KUKA KRL program: MyProgram_030().src

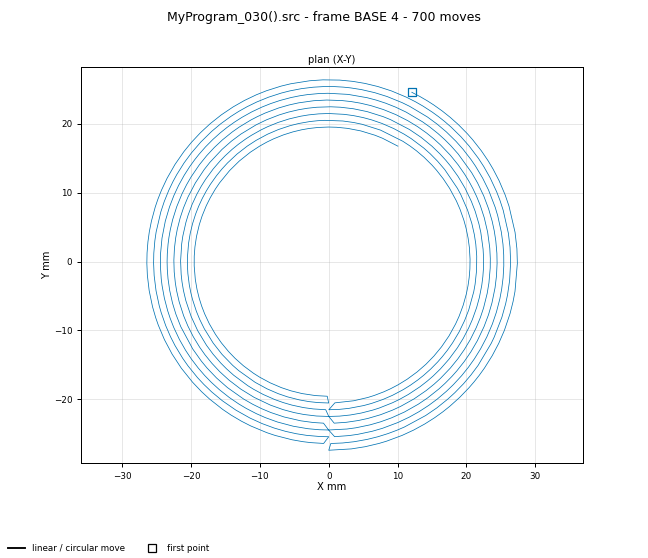
[picture p0: tool path of MyProgram_030().src in frame BASE 4, 700 of 700 moves have a stored position in this frame; points joined in program order, loops and branches not executed]
&ACCESS RVP
&REL 1
&PARAM TEMPLATE = C:\KRC\Roboter\Template\vorgabe
&PARAM EDITMASK = *
DEF MyProgram_030()
; ---- Setting reference (Base) ----
$BASE = BASE_DATA[4]

; --------------------------
; ---- Setting tool (TCP) ----
$TOOL = TOOL_DATA[3]
; --------------------------

$VEL.CP = VEL_APROX_PRINT
Startdeposition()
$VEL.CP = VEL_PRINT
LIN {X 12.0703,Y 24.5921,Z 59,A 55.5267,B 24.8071,C -3.2024,E1 25.0724,E2 -692.837} C_DIS
LIN {X 13.2585,Y 23.9727,Z 59,A 52.8062,B 24.8075,C -3.1996,E1 25.0791,E2 -690.1175} C_DIS
LIN {X 14.3009,Y 23.3657,Z 59,A 50.2739,B 24.8079,C -3.1959,E1 25.0852,E2 -687.5843} C_DIS
LIN {X 15.2376,Y 22.7662,Z 59,A 47.9776,B 24.8083,C -3.1926,E1 25.0906,E2 -685.2878} C_DIS
LIN {X 16.4743,Y 21.887,Z 59,A 44.3349,B 24.8096,C -3.1823,E1 25.0988,E2 -681.6335} C_DIS
LIN {X 17.6466,Y 20.9541,Z 59,A 41.1874,B 24.8103,C -3.1764,E1 25.1056,E2 -678.484} C_DIS
LIN {X 18.834,Y 19.8936,Z 59,A 38.0345,B 24.8108,C -3.1718,E1 25.112,E2 -675.333} C_DIS
LIN {X 20.1281,Y 18.5822,Z 59,A 34.6982,B 24.8111,C -3.1694,E1 25.1185,E2 -672.0053} C_DIS
LIN {X 20.8979,Y 17.7129,Z 59,A 31.723,B 24.8125,C -3.1578,E1 25.1239,E2 -669.0162} C_DIS
LIN {X 22.1576,Y 16.1093,Z 59,A 27.8177,B 24.8132,C -3.1518,E1 25.1305,E2 -665.1153} C_DIS
LIN {X 23.1629,Y 14.6275,Z 59,A 23.876,B 24.8146,C -3.1402,E1 25.1366,E2 -661.1657} C_DIS
LIN {X 23.8751,Y 13.4329,Z 59,A 20.9616,B 24.8155,C -3.1326,E1 25.1406,E2 -658.2484} C_DIS
LIN {X 24.7489,Y 11.7454,Z 59,A 16.9906,B 24.8168,C -3.1219,E1 25.1455,E2 -654.2731} C_DIS
LIN {X 25.6294,Y 9.6744,Z 59,A 11.8386,B 24.8189,C -3.1034,E1 25.1509,E2 -649.1059} C_DIS
LIN {X 26.1818,Y 8.0609,Z 59,A 7.6845,B 24.8209,C -3.0861,E1 25.1543,E2 -644.9344} C_DIS
LIN {X 27.0615,Y 4.2601,Z 59,A 1.2889,B 24.8214,C -3.0826,E1 25.158,E2 -638.5678} C_DIS
LIN {X 27.3301,Y 1.8802,Z 59,A -5.3272,B 24.8254,C -3.0478,E1 25.1597,E2 -631.9085} C_DIS
LIN {X 27.3946,Y -0.2461,Z 59,A -10.1009,B 24.8274,C -3.0301,E1 25.1596,E2 -627.1211} C_DIS
LIN {X 27.0526,Y -4.3175,Z 59,A -16.9925,B 24.8282,C -3.0233,E1 25.1575,E2 -620.2542} C_DIS
LIN {X 26.776,Y -5.7881,Z 59,A -20.1318,B 24.8293,C -3.0135,E1 25.1557,E2 -617.11} C_DIS
LIN {X 26.3337,Y -7.5501,Z 59,A -23.8827,B 24.8306,C -3.0024,E1 25.153,E2 -613.3544} C_DIS
LIN {X 25.5178,Y -9.9656,Z 59,A -30.3379,B 24.8339,C -2.973,E1 25.1468,E2 -606.8657} C_DIS
LIN {X 24.6926,Y -11.8634,Z 59,A -33.9623,B 24.8344,C -2.9686,E1 25.1426,E2 -603.2505} C_DIS
LIN {X 23.7431,Y -13.6635,Z 59,A -37.9233,B 24.8353,C -2.9601,E1 25.1372,E2 -599.2899} C_DIS
LIN {X 22.6158,Y -15.4593,Z 59,A -41.7608,B 24.8359,C -2.9549,E1 25.1314,E2 -595.4595} C_DIS
LIN {X 21.8598,Y -16.5112,Z 59,A -44.5998,B 24.8369,C -2.9462,E1 25.1267,E2 -592.6136} C_DIS
LIN {X 21.1214,Y -17.4459,Z 59,A -47.2368,B 24.8378,C -2.9381,E1 25.1221,E2 -589.9696} C_DIS
LIN {X 20.3552,Y -18.3341,Z 59,A -49.8939,B 24.8387,C -2.9297,E1 25.1172,E2 -587.3044} C_DIS
LIN {X 18.9974,Y -19.7374,Z 59,A -54.0497,B 24.8399,C -2.9192,E1 25.1089,E2 -583.1413} C_DIS
LIN {X 17.5559,Y -21.03,Z 59,A -57.5749,B 24.8402,C -2.9161,E1 25.1015,E2 -579.6227} C_DIS
LIN {X 16.5729,Y -21.8133,Z 59,A -60.5172,B 24.8412,C -2.9071,E1 25.095,E2 -576.6699} C_DIS
LIN {X 15.3797,Y -22.6701,Z 59,A -63.5679,B 24.8418,C -2.9013,E1 25.088,E2 -573.6159} C_DIS
LIN {X 13.9552,Y -23.5737,Z 59,A -67.0294,B 24.8425,C -2.8956,E1 25.0798,E2 -570.1517} C_DIS
LIN {X 12.3253,Y -24.4654,Z 59,A -71.4342,B 24.8438,C -2.8836,E1 25.0689,E2 -565.7309} C_DIS
LIN {X 10.6544,Y -25.2378,Z 59,A -75.2339,B 24.8443,C -2.8786,E1 25.0591,E2 -561.9284} C_DIS
LIN {X 8.4028,Y -26.0738,Z 59,A -79.4966,B 24.8442,C -2.8801,E1 25.0479,E2 -557.6779} C_DIS
LIN {X 7.3143,Y -26.4001,Z 59,A -82.2216,B 24.8448,C -2.874,E1 25.0406,E2 -554.943} C_DIS
LIN {X 5.3186,Y -26.8736,Z 59,A -86.9065,B 24.8456,C -2.8663,E1 25.0278,E2 -550.246} C_DIS
LIN {X 3.2945,Y -27.1959,Z 59,A -91.5499,B 24.8463,C -2.8601,E1 25.0149,E2 -545.5918} C_DIS
LIN {X 0.0059,Y -27.3922,Z 59,A -95.1262,B 24.8432,C -2.889,E1 25.0051,E2 -542.0856} C_DIS
Enddeposition()
LIN {X 0.0059,Y -27.3922,Z 59,A -95.1262,B 24.8432,C -2.889,E1 25.0051,E2 -542.0856} C_DIS
Startdeposition()
$VEL.CP = VEL_PRINT
LIN {X 0.2993,Y -26.4122,Z 59,A -95.4906,B 24.8424,C -2.8963,E1 25.0042,E2 -541.7387} C_DIS
LIN {X 2.0234,Y -26.3363,Z 59,A -91.3024,B 24.8418,C -2.902,E1 25.0159,E2 -545.9388} C_DIS
LIN {X 3.7058,Y -26.1526,Z 59,A -87.6758,B 24.8415,C -2.9039,E1 25.0259,E2 -549.5669} C_DIS
LIN {X 5.5925,Y -25.8151,Z 59,A -83.5455,B 24.8412,C -2.9071,E1 25.0372,E2 -553.6998} C_DIS
LIN {X 7.1324,Y -25.4327,Z 59,A -80.3986,B 24.8412,C -2.9077,E1 25.0457,E2 -556.8432} C_DIS
LIN {X 8.5837,Y -24.9799,Z 59,A -77.2197,B 24.8408,C -2.9104,E1 25.0541,E2 -560.0224} C_DIS
LIN {X 9.8795,Y -24.4969,Z 59,A -74.2469,B 24.8404,C -2.9141,E1 25.0619,E2 -562.9976} C_DIS
LIN {X 10.9902,Y -24.019,Z 59,A -70.5185,B 24.8387,C -2.9297,E1 25.0714,E2 -566.7536} C_DIS
LIN {X 14.0844,Y -22.3457,Z 59,A -63.6414,B 24.8381,C -2.9349,E1 25.088,E2 -573.6223} C_DIS
LIN {X 15.6927,Y -21.2472,Z 59,A -59.3824,B 24.8372,C -2.9437,E1 25.0977,E2 -577.8875} C_DIS
LIN {X 17.2836,Y -19.9745,Z 59,A -55.1439,B 24.8363,C -2.9513,E1 25.1068,E2 -582.1276} C_DIS
LIN {X 18.3176,Y -19.0305,Z 59,A -51.8874,B 24.8353,C -2.9608,E1 25.1135,E2 -585.3932} C_DIS
LIN {X 19.5777,Y -17.7319,Z 59,A -48.5226,B 24.8349,C -2.9639,E1 25.1199,E2 -588.7508} C_DIS
LIN {X 20.6509,Y -16.4691,Z 59,A -44.3687,B 24.8332,C -2.9795,E1 25.1273,E2 -592.9225} C_DIS
LIN {X 21.6906,Y -15.0734,Z 59,A -39.8108,B 24.831,C -2.9989,E1 25.1346,E2 -597.5039} C_DIS
LIN {X 23.5983,Y -11.8668,Z 59,A -33.2485,B 24.8304,C -3.0036,E1 25.1435,E2 -604.0433} C_DIS
LIN {X 24.0437,Y -10.9355,Z 59,A -29.9775,B 24.8283,C -3.0224,E1 25.1474,E2 -607.3412} C_DIS
LIN {X 25.1471,Y -8.0821,Z 59,A -23.9084,B 24.8268,C -3.0356,E1 25.1531,E2 -613.4073} C_DIS
LIN {X 25.6939,Y -6.1255,Z 59,A -20.1339,B 24.8261,C -3.0415,E1 25.1558,E2 -617.1743} C_DIS
LIN {X 25.9662,Y -4.8406,Z 59,A -17.0738,B 24.8248,C -3.0529,E1 25.1574,E2 -620.2434} C_DIS
LIN {X 26.2688,Y -2.7644,Z 59,A -11.7155,B 24.822,C -3.0768,E1 25.1593,E2 -625.6269} C_DIS
LIN {X 26.4161,Y -0.0885,Z 59,A -6.3971,B 24.8206,C -3.089,E1 25.1598,E2 -630.9423} C_DIS
LIN {X 26.3302,Y 2.1008,Z 59,A -1.385,B 24.8185,C -3.1069,E1 25.1589,E2 -635.967} C_DIS
LIN {X 26.0901,Y 4.1243,Z 59,A 3.4136,B 24.8164,C -3.1249,E1 25.1569,E2 -640.7802} C_DIS
LIN {X 25.3421,Y 7.4472,Z 59,A 9.6225,B 24.8155,C -3.1328,E1 25.1528,E2 -646.9719} C_DIS
LIN {X 24.8708,Y 8.8956,Z 59,A 13.13,B 24.814,C -3.1447,E1 25.1496,E2 -650.4879} C_DIS
LIN {X 24.3916,Y 10.136,Z 59,A 16.1141,B 24.8129,C -3.154,E1 25.1465,E2 -653.4776} C_DIS
LIN {X 23.4463,Y 12.1643,Z 59,A 21.2351,B 24.811,C -3.1702,E1 25.1401,E2 -658.6096} C_DIS
LIN {X 22.5009,Y 13.8356,Z 59,A 25.1058,B 24.8101,C -3.1776,E1 25.1346,E2 -662.4779} C_DIS
LIN {X 21.7431,Y 14.9976,Z 59,A 28.195,B 24.8091,C -3.1859,E1 25.1298,E2 -665.5716} C_DIS
LIN {X 20.3882,Y 16.7935,Z 59,A 32.3345,B 24.8087,C -3.189,E1 25.1227,E2 -669.6989} C_DIS
LIN {X 19.2048,Y 18.1348,Z 59,A 37.0991,B 24.8065,C -3.2072,E1 25.1137,E2 -674.4856} C_DIS
LIN {X 17.7872,Y 19.5274,Z 59,A 40.7472,B 24.8064,C -3.2086,E1 25.1063,E2 -678.1221} C_DIS
LIN {X 16.8166,Y 20.3691,Z 59,A 43.3718,B 24.806,C -3.2121,E1 25.1007,E2 -680.7447} C_DIS
LIN {X 15.9526,Y 21.0528,Z 59,A 45.8165,B 24.8054,C -3.2169,E1 25.0953,E2 -683.1917} C_DIS
LIN {X 15.0479,Y 21.7084,Z 59,A 48.563,B 24.8045,C -3.2242,E1 25.089,E2 -685.9461} C_DIS
LIN {X 13.6911,Y 22.5887,Z 59,A 51.7172,B 24.8043,C -3.2258,E1 25.0816,E2 -689.094} C_DIS
LIN {X 12.6011,Y 23.2143,Z 59,A 54.6274,B 24.8036,C -3.2313,E1 25.0745,E2 -692.0088} C_DIS
LIN {X 11.2915,Y 23.8787,Z 59,A 58.2581,B 24.8026,C -3.2396,E1 25.0653,E2 -695.6495} C_DIS
LIN {X 9.1052,Y 24.7944,Z 59,A 62.8093,B 24.8027,C -3.2388,E1 25.0536,E2 -700.1886} C_DIS
LIN {X 7.1428,Y 25.4295,Z 59,A 67.9203,B 24.8016,C -3.2481,E1 25.0399,E2 -705.3127} C_DIS
LIN {X 5.2719,Y 25.8825,Z 59,A 71.5741,B 24.8019,C -3.2452,E1 25.03,E2 -708.9548} C_DIS
LIN {X 3.4856,Y 26.183,Z 59,A 75.855,B 24.8014,C -3.2495,E1 25.0181,E2 -713.242} C_DIS
LIN {X 1.5804,Y 26.3662,Z 59,A 80.1393,B 24.8012,C -3.2508,E1 25.0062,E2 -717.5274} C_DIS
LIN {X -0.8248,Y 26.401,Z 59,A 85.1216,B 24.8016,C -3.2477,E1 24.9923,E2 -722.5021} C_DIS
LIN {X -2.7464,Y 26.2707,Z 59,A 89.7241,B 24.8014,C -3.2493,E1 24.9795,E2 -727.1108} C_DIS
LIN {X -5.5246,Y 25.8296,Z 59,A 94.8895,B 24.8029,C -3.2373,E1 24.9654,E2 -732.2526} C_DIS
LIN {X -6.9255,Y 25.4898,Z 59,A 98.7337,B 24.8026,C -3.2398,E1 24.9549,E2 -736.1086} C_DIS
LIN {X -9.0534,Y 24.8138,Z 59,A 103.2055,B 24.8036,C -3.2313,E1 24.9431,E2 -740.5684} C_DIS
LIN {X -10.5209,Y 24.2282,Z 59,A 106.666,B 24.8042,C -3.2268,E1 24.9342,E2 -744.0261} C_DIS
LIN {X -12.2342,Y 23.4094,Z 59,A 111.5552,B 24.8042,C -3.2259,E1 24.922,E2 -748.9262} C_DIS
LIN {X -13.8723,Y 22.4777,Z 59,A 115.2888,B 24.8055,C -3.2162,E1 24.9131,E2 -752.648} C_DIS
LIN {X -15.6046,Y 21.3117,Z 59,A 119.666,B 24.8067,C -3.2063,E1 24.9031,E2 -757.0166} C_DIS
LIN {X -17.2144,Y 20.034,Z 59,A 124.0536,B 24.8079,C -3.1963,E1 24.8937,E2 -761.397} C_DIS
LIN {X -18.6321,Y 18.7227,Z 59,A 128.3146,B 24.809,C -3.1872,E1 24.8851,E2 -765.6537} C_DIS
LIN {X -19.9447,Y 17.3177,Z 59,A 132.7337,B 24.81,C -3.1785,E1 24.8769,E2 -770.0719} C_DIS
LIN {X -21.0478,Y 15.9592,Z 59,A 136.4195,B 24.8113,C -3.1681,E1 24.8706,E2 -773.75} C_DIS
LIN {X -22.3201,Y 14.1253,Z 59,A 141.3942,B 24.8127,C -3.1558,E1 24.8629,E2 -778.7202} C_DIS
LIN {X -23.4768,Y 12.1054,Z 59,A 146.3251,B 24.8145,C -3.1408,E1 24.8563,E2 -783.6412} C_DIS
LIN {X -24.2947,Y 10.3665,Z 59,A 150.5155,B 24.8159,C -3.1287,E1 24.8515,E2 -787.8257} C_DIS
LIN {X -24.82,Y 9.0365,Z 59,A 153.5544,B 24.8171,C -3.1191,E1 24.8486,E2 -790.8587} C_DIS
LIN {X -25.2006,Y 7.9134,Z 59,A 156.3755,B 24.8178,C -3.1127,E1 24.8462,E2 -793.6808} C_DIS
LIN {X -25.7517,Y 5.875,Z 59,A 160.3956,B 24.8199,C -3.0955,E1 24.8434,E2 -797.683} C_DIS
LIN {X -26.0575,Y 4.3243,Z 59,A 163.709,B 24.8212,C -3.0842,E1 24.8417,E2 -800.989} C_DIS
LIN {X -26.2568,Y 2.8758,Z 59,A 167.4625,B 24.8219,C -3.0776,E1 24.8404,E2 -804.7491} C_DIS
LIN {X -26.3843,Y 1.2532,Z 59,A 170.8053,B 24.8233,C -3.0655,E1 24.8399,E2 -808.0831} C_DIS
LIN {X -26.4138,Y -0.2385,Z 59,A 174.1449,B 24.8244,C -3.056,E1 24.8399,E2 -811.42} C_DIS
LIN {X -26.3409,Y -1.9594,Z 59,A 178.5048,B 24.8254,C -3.0481,E1 24.8406,E2 -815.787} C_DIS
LIN {X -26.0758,Y -4.2115,Z 59,A -176.6427,B 24.8271,C -3.0327,E1 24.8425,E2 -820.6316} C_DIS
LIN {X -25.5842,Y -6.5683,Z 59,A -171.8967,B 24.8292,C -3.0142,E1 24.8455,E2 -825.3613} C_DIS
LIN {X -25.1234,Y -8.1552,Z 59,A -168.5165,B 24.8305,C -3.0026,E1 24.8482,E2 -828.7332} C_DIS
LIN {X -24.7509,Y -9.2239,Z 59,A -165.4952,B 24.831,C -2.999,E1 24.8511,E2 -831.7628} C_DIS
LIN {X -23.8641,Y -11.3221,Z 59,A -160.9304,B 24.8328,C -2.983,E1 24.8563,E2 -836.3145} C_DIS
LIN {X -22.7493,Y -13.4226,Z 59,A -154.8114,B 24.8336,C -2.9756,E1 24.8646,E2 -842.4478} C_DIS
LIN {X -21.4033,Y -15.4784,Z 59,A -149.6935,B 24.8352,C -2.9612,E1 24.8728,E2 -847.5566} C_DIS
LIN {X -19.7669,Y -17.5208,Z 59,A -144.5853,B 24.8371,C -2.9446,E1 24.8819,E2 -852.6486} C_DIS
LIN {X -18.4746,Y -18.8784,Z 59,A -140.343,B 24.8379,C -2.9374,E1 24.8902,E2 -856.8918} C_DIS
LIN {X -17.2945,Y -19.9651,Z 59,A -136.6082,B 24.8384,C -2.9326,E1 24.898,E2 -860.6299} C_DIS
LIN {X -15.3939,Y -21.4644,Z 59,A -131.6256,B 24.8396,C -2.9217,E1 24.9091,E2 -865.6044} C_DIS
LIN {X -14.1777,Y -22.2866,Z 59,A -128.37,B 24.8401,C -2.9174,E1 24.9167,E2 -868.8603} C_DIS
LIN {X -12.6662,Y -23.1788,Z 59,A -124.9787,B 24.841,C -2.9091,E1 24.9249,E2 -872.2419} C_DIS
LIN {X -11.3388,Y -23.8563,Z 59,A -120.8569,B 24.8406,C -2.9123,E1 24.9353,E2 -876.3819} C_DIS
LIN {X -8.9797,Y -24.8407,Z 59,A -116.0784,B 24.8419,C -2.9009,E1 24.9476,E2 -881.1437} C_DIS
LIN {X -7.7901,Y -25.2388,Z 59,A -112.6547,B 24.8415,C -2.9047,E1 24.9568,E2 -884.5825} C_DIS
LIN {X -5.3326,Y -25.87,Z 59,A -107.6975,B 24.8423,C -2.8974,E1 24.9702,E2 -889.5289} C_DIS
LIN {X -3.7588,Y -26.1451,Z 59,A -104.4193,B 24.8425,C -2.8948,E1 24.9793,E2 -892.804} C_DIS
LIN {X -2.5933,Y -26.286,Z 59,A -101.7053,B 24.8425,C -2.896,E1 24.9868,E2 -895.5224} C_DIS
LIN {X -0.7369,Y -26.4036,Z 59,A -97.345,B 24.8421,C -2.8993,E1 24.999,E2 -899.8916} C_DIS
LIN {X -0.7369,Y -26.4036,Z 59,A -97.345,B 24.8421,C -2.8993,E1 24.999,E2 -899.8916} C_DIS
Enddeposition()
LIN {X 0.0029,Y -25.4285,Z 59,A -96.2561,B 24.8407,C -2.9118,E1 25.0021,E2 -901.0102} C_DIS
Startdeposition()
$VEL.CP = VEL_PRINT
LIN {X -1.2097,Y -25.4043,Z 59,A -100.6786,B 24.8423,C -2.8969,E1 24.9897,E2 -896.5516} C_DIS
LIN {X -3.1937,Y -25.2319,Z 59,A -104.8094,B 24.842,C -2.9002,E1 24.9782,E2 -892.4263} C_DIS
LIN {X -4.7198,Y -24.9913,Z 59,A -108.5025,B 24.842,C -2.8996,E1 24.968,E2 -888.7281} C_DIS
LIN {X -6.2671,Y -24.649,Z 59,A -112.0147,B 24.8418,C -2.9018,E1 24.9585,E2 -885.2165} C_DIS
LIN {X -7.9099,Y -24.1718,Z 59,A -116.0499,B 24.8416,C -2.9031,E1 24.9477,E2 -881.1775} C_DIS
LIN {X -9.6577,Y -23.528,Z 59,A -120.3493,B 24.8413,C -2.9062,E1 24.9365,E2 -876.8763} C_DIS
LIN {X -11.4145,Y -22.728,Z 59,A -124.859,B 24.8409,C -2.9101,E1 24.9252,E2 -872.3642} C_DIS
LIN {X -13.4858,Y -21.5633,Z 59,A -129.8541,B 24.8398,C -2.92,E1 24.9132,E2 -867.3777} C_DIS
LIN {X -15.451,Y -20.2019,Z 59,A -135.9915,B 24.8393,C -2.9239,E1 24.8993,E2 -861.2282} C_DIS
LIN {X -16.9968,Y -18.9197,Z 59,A -139.5957,B 24.8378,C -2.9383,E1 24.8917,E2 -857.6442} C_DIS
LIN {X -18.1286,Y -17.8381,Z 59,A -143.2487,B 24.8371,C -2.9446,E1 24.8844,E2 -853.991} C_DIS
LIN {X -19.0676,Y -16.831,Z 59,A -146.794,B 24.8366,C -2.9486,E1 24.8778,E2 -850.4395} C_DIS
LIN {X -20.437,Y -15.1385,Z 59,A -151.2321,B 24.835,C -2.9628,E1 24.8702,E2 -846.0143} C_DIS
LIN {X -21.1995,Y -14.0509,Z 59,A -154.7216,B 24.8345,C -2.9673,E1 24.8647,E2 -842.5182} C_DIS
LIN {X -22.3187,Y -12.1953,Z 59,A -159.217,B 24.8329,C -2.9821,E1 24.8584,E2 -838.0349} C_DIS
LIN {X -22.9714,Y -10.9156,Z 59,A -162.464,B 24.8319,C -2.9908,E1 24.8544,E2 -834.7911} C_DIS
LIN {X -23.6766,Y -9.2878,Z 59,A -167.013,B 24.831,C -2.9989,E1 24.8496,E2 -830.2364} C_DIS
LIN {X -24.3384,Y -7.3808,Z 59,A -170.8482,B 24.829,C -3.0159,E1 24.8463,E2 -826.4199} C_DIS
LIN {X -24.6196,Y -6.3814,Z 59,A -173.8342,B 24.8286,C -3.0194,E1 24.8441,E2 -823.4249} C_DIS
LIN {X -25.0782,Y -4.2337,Z 59,A -178.4371,B 24.8267,C -3.0361,E1 24.8417,E2 -818.8348} C_DIS
LIN {X -25.3526,Y -2.0218,Z 59,A 175.9685,B 24.8253,C -3.0486,E1 24.84,E2 -813.2369} C_DIS
LIN {X -25.4329,Y -0.2384,Z 59,A 172.5211,B 24.8235,C -3.064,E1 24.8398,E2 -809.8056} C_DIS
LIN {X -25.404,Y 1.2223,Z 59,A 168.955,B 24.8225,C -3.0729,E1 24.8401,E2 -806.2393} C_DIS
LIN {X -25.2509,Y 3.0384,Z 59,A 164.8825,B 24.821,C -3.0859,E1 24.8413,E2 -802.1735} C_DIS
LIN {X -25.0675,Y 4.2978,Z 59,A 161.1273,B 24.8205,C -3.0903,E1 24.843,E2 -798.4065} C_DIS
LIN {X -24.3856,Y 7.2226,Z 59,A 155.1133,B 24.8176,C -3.1149,E1 24.8472,E2 -792.4164} C_DIS
LIN {X -23.8897,Y 8.725,Z 59,A 151.608,B 24.8163,C -3.1259,E1 24.8504,E2 -788.9175} C_DIS
LIN {X -23.2327,Y 10.3479,Z 59,A 147.5318,B 24.815,C -3.1368,E1 24.8549,E2 -784.8449} C_DIS
LIN {X -22.6279,Y 11.6114,Z 59,A 144.7317,B 24.8137,C -3.1478,E1 24.8583,E2 -782.056} C_DIS
LIN {X -22.0725,Y 12.635,Z 59,A 141.8531,B 24.813,C -3.1538,E1 24.8622,E2 -779.1766} C_DIS
LIN {X -21.0151,Y 14.3254,Z 59,A 137.0769,B 24.8117,C -3.1644,E1 24.8695,E2 -774.402} C_DIS
LIN {X -19.9531,Y 15.7706,Z 59,A 132.857,B 24.8106,C -3.1739,E1 24.8767,E2 -770.1846} C_DIS
LIN {X -18.5886,Y 17.3585,Z 59,A 128.2533,B 24.8091,C -3.1861,E1 24.8852,E2 -765.5896} C_DIS
LIN {X -17.0144,Y 18.9039,Z 59,A 123.8457,B 24.8073,C -3.2008,E1 24.8941,E2 -761.1989} C_DIS
LIN {X -15.7044,Y 20.0049,Z 59,A 119.4167,B 24.8068,C -3.2055,E1 24.9037,E2 -756.7644} C_DIS
LIN {X -14.1904,Y 21.1064,Z 59,A 115.1874,B 24.8058,C -3.2136,E1 24.9134,E2 -752.54} C_DIS
LIN {X -13.0773,Y 21.8138,Z 59,A 112.2766,B 24.8051,C -3.2193,E1 24.9203,E2 -749.6339} C_DIS
LIN {X -11.8565,Y 22.5003,Z 59,A 109.2672,B 24.8043,C -3.2254,E1 24.9277,E2 -746.6307} C_DIS
LIN {X -10.4592,Y 23.1827,Z 59,A 105.568,B 24.8039,C -3.2294,E1 24.937,E2 -742.9316} C_DIS
LIN {X -8.7401,Y 23.8841,Z 59,A 101.273,B 24.8033,C -3.234,E1 24.9482,E2 -738.6386} C_DIS
LIN {X -6.8909,Y 24.4817,Z 59,A 97.3409,B 24.8023,C -3.242,E1 24.9587,E2 -734.7187} C_DIS
LIN {X -5.6559,Y 24.7962,Z 59,A 94.5218,B 24.8019,C -3.245,E1 24.9663,E2 -731.903} C_DIS
LIN {X -3.9707,Y 25.1214,Z 59,A 90.0778,B 24.8021,C -3.2435,E1 24.9786,E2 -727.4509} C_DIS
LIN {X -2.2699,Y 25.3317,Z 59,A 86.6573,B 24.8015,C -3.2489,E1 24.988,E2 -724.0413} C_DIS
LIN {X -0.7618,Y 25.4217,Z 59,A 83.0977,B 24.8015,C -3.2489,E1 24.998,E2 -720.4807} C_DIS
LIN {X 0.824,Y 25.4198,Z 59,A 79.4962,B 24.8015,C -3.2491,E1 25.008,E2 -716.8803} C_DIS
LIN {X 2.1249,Y 25.3444,Z 59,A 76.9034,B 24.8011,C -3.2518,E1 25.0152,E2 -714.2952} C_DIS
LIN {X 3.1883,Y 25.2326,Z 59,A 74.4415,B 24.8012,C -3.251,E1 25.022,E2 -711.833} C_DIS
LIN {X 4.7781,Y 24.9802,Z 59,A 70.3399,B 24.8019,C -3.2457,E1 25.0333,E2 -707.7231} C_DIS
LIN {X 6.6882,Y 24.5378,Z 59,A 65.8684,B 24.8022,C -3.2427,E1 25.0454,E2 -703.2512} C_DIS
LIN {X 8.4653,Y 23.983,Z 59,A 61.58,B 24.8027,C -3.2384,E1 25.0568,E2 -698.961} C_DIS
LIN {X 10.6559,Y 23.0928,Z 59,A 57.0526,B 24.8025,C -3.2403,E1 25.0684,E2 -694.4489} C_DIS
LIN {X 11.7518,Y 22.5552,Z 59,A 53.0766,B 24.8044,C -3.2253,E1 25.0783,E2 -690.4481} C_DIS
LIN {X 14.3371,Y 21.0071,Z 59,A 47.2176,B 24.8044,C -3.2242,E1 25.0921,E2 -684.6052} C_DIS
LIN {X 15.7416,Y 19.9761,Z 59,A 43.0326,B 24.8056,C -3.2148,E1 25.1014,E2 -680.4132} C_DIS
LIN {X 17.0881,Y 18.8377,Z 59,A 39.0137,B 24.8066,C -3.2067,E1 25.1099,E2 -676.3911} C_DIS
LIN {X 18.4791,Y 17.4749,Z 59,A 34.6879,B 24.8076,C -3.1982,E1 25.1183,E2 -672.0636} C_DIS
LIN {X 19.4973,Y 16.3312,Z 59,A 31.2503,B 24.8086,C -3.1906,E1 25.1246,E2 -668.6236} C_DIS
LIN {X 20.6767,Y 14.8086,Z 59,A 27.5181,B 24.809,C -3.1868,E1 25.1308,E2 -664.9001} C_DIS
LIN {X 21.3209,Y 13.8654,Z 59,A 24.4553,B 24.8104,C -3.1752,E1 25.1356,E2 -661.8249} C_DIS
LIN {X 22.3589,Y 12.1212,Z 59,A 19.8289,B 24.8119,C -3.1626,E1 25.142,E2 -657.1928} C_DIS
LIN {X 23.2157,Y 10.3861,Z 59,A 14.9669,B 24.814,C -3.1452,E1 25.1477,E2 -652.3157} C_DIS
LIN {X 24.1822,Y 7.8781,Z 59,A 9.8931,B 24.8148,C -3.1388,E1 25.1525,E2 -647.2552} C_DIS
LIN {X 24.5451,Y 6.661,Z 59,A 6.4065,B 24.8166,C -3.1233,E1 25.1552,E2 -643.7519} C_DIS
LIN {X 25.0652,Y 4.311,Z 59,A 1.43,B 24.8179,C -3.112,E1 25.1579,E2 -638.7777} C_DIS
LIN {X 25.3071,Y 2.5294,Z 59,A -2.4181,B 24.8191,C -3.1019,E1 25.1592,E2 -634.9283} C_DIS
LIN {X 25.4149,Y 0.9636,Z 59,A -5.996,B 24.8204,C -3.0904,E1 25.1597,E2 -631.3445} C_DIS
LIN {X 25.4261,Y -0.5978,Z 59,A -9.6939,B 24.822,C -3.0774,E1 25.1597,E2 -627.6377} C_DIS
LIN {X 25.3255,Y -2.3358,Z 59,A -13.4112,B 24.8231,C -3.0675,E1 25.1589,E2 -623.919} C_DIS
LIN {X 25.1224,Y -3.9642,Z 59,A -16.7111,B 24.8239,C -3.0605,E1 25.1576,E2 -620.6221} C_DIS
LIN {X 24.8548,Y -5.3931,Z 59,A -20.5219,B 24.8258,C -3.0442,E1 25.1555,E2 -616.7949} C_DIS
LIN {X 24.3534,Y -7.3318,Z 59,A -24.6298,B 24.8269,C -3.035,E1 25.1525,E2 -612.6887} C_DIS
LIN {X 23.7604,Y -9.0714,Z 59,A -29.4018,B 24.8291,C -3.0154,E1 25.1479,E2 -607.897} C_DIS
LIN {X 22.9618,Y -10.9359,Z 59,A -33.5305,B 24.8301,C -3.0069,E1 25.1432,E2 -603.7707} C_DIS
LIN {X 22.0581,Y -12.6603,Z 59,A -38.2666,B 24.8319,C -2.9905,E1 25.1368,E2 -599.0206} C_DIS
LIN {X 21.1541,Y -14.1193,Z 59,A -41.4854,B 24.8323,C -2.9871,E1 25.132,E2 -595.8098} C_DIS
LIN {X 20.2829,Y -15.3442,Z 59,A -45.0898,B 24.8336,C -2.9757,E1 25.126,E2 -592.1959} C_DIS
LIN {X 19.2887,Y -16.5772,Z 59,A -48.6687,B 24.8346,C -2.9665,E1 25.1196,E2 -588.6116} C_DIS
LIN {X 18.0945,Y -17.8725,Z 59,A -52.0169,B 24.8349,C -2.9636,E1 25.1132,E2 -585.2711} C_DIS
LIN {X 17.1,Y -18.8266,Z 59,A -55.8808,B 24.8366,C -2.9484,E1 25.1053,E2 -581.3869} C_DIS
LIN {X 15.7614,Y -19.9605,Z 59,A -59.4997,B 24.8372,C -2.9434,E1 25.0975,E2 -577.7699} C_DIS
LIN {X 14.5389,Y -20.8677,Z 59,A -63.1802,B 24.8382,C -2.9339,E1 25.0891,E2 -574.0798} C_DIS
LIN {X 13.1364,Y -21.778,Z 59,A -66.6228,B 24.8386,C -2.9303,E1 25.081,E2 -570.6395} C_DIS
LIN {X 11.6819,Y -22.5917,Z 59,A -70.6854,B 24.8397,C -2.9209,E1 25.071,E2 -566.5663} C_DIS
LIN {X 10.0323,Y -23.3706,Z 59,A -74.9974,B 24.8406,C -2.9128,E1 25.0599,E2 -562.2458} C_DIS
LIN {X 7.8031,Y -24.2065,Z 59,A -80.0293,B 24.841,C -2.9093,E1 25.0467,E2 -557.2156} C_DIS
LIN {X 6.3093,Y -24.6381,Z 59,A -83.7277,B 24.8416,C -2.9039,E1 25.0367,E2 -553.5102} C_DIS
LIN {X 4.2259,Y -25.0796,Z 59,A -88.1915,B 24.8416,C -2.903,E1 25.0245,E2 -549.0496} C_DIS
LIN {X 2.9311,Y -25.2637,Z 59,A -91.349,B 24.8421,C -2.8993,E1 25.0157,E2 -545.8858} C_DIS
LIN {X 0.8535,Y -25.4189,Z 59,A -96.2183,B 24.8424,C -2.8959,E1 25.0021,E2 -541.0102} C_DIS
LIN {X 0.8535,Y -25.4189,Z 59,A -96.2183,B 24.8424,C -2.8959,E1 25.0021,E2 -541.0102} C_DIS
Enddeposition()
LIN {X -0.0174,Y -24.4501,Z 59,A -95.7637,B 24.8383,C -2.9331,E1 25.0036,E2 -541.5533} C_DIS
Startdeposition()
$VEL.CP = VEL_PRINT
LIN {X 2.6429,Y -24.3091,Z 59,A -90.1866,B 24.8387,C -2.9301,E1 25.0191,E2 -547.1206} C_DIS
LIN {X 3.9479,Y -24.1317,Z 59,A -86.4823,B 24.8378,C -2.9377,E1 25.0294,E2 -550.8396} C_DIS
LIN {X 6.0113,Y -23.7019,Z 59,A -81.8333,B 24.8376,C -2.9396,E1 25.0421,E2 -555.4867} C_DIS
LIN {X 7.5479,Y -23.2583,Z 59,A -78.0587,B 24.8371,C -2.9441,E1 25.0521,E2 -559.2652} C_DIS
LIN {X 9.1385,Y -22.6805,Z 59,A -73.9004,B 24.8363,C -2.9512,E1 25.063,E2 -563.4314} C_DIS
LIN {X 10.9875,Y -21.8449,Z 59,A -68.8652,B 24.8352,C -2.9614,E1 25.0757,E2 -568.4775} C_DIS
LIN {X 13.0092,Y -20.7047,Z 59,A -63.9982,B 24.8347,C -2.9653,E1 25.0874,E2 -573.3389} C_DIS
LIN {X 14.3498,Y -19.7992,Z 59,A -60.0893,B 24.8338,C -2.974,E1 25.0963,E2 -577.255} C_DIS
LIN {X 16.006,Y -18.486,Z 59,A -55.2834,B 24.8327,C -2.9831,E1 25.1067,E2 -582.0643} C_DIS
LIN {X 16.9104,Y -17.6625,Z 59,A -52.5113,B 24.8321,C -2.9887,E1 25.1124,E2 -584.8382} C_DIS
LIN {X 17.8829,Y -16.6767,Z 59,A -49.5074,B 24.8315,C -2.994,E1 25.1182,E2 -587.8416} C_DIS
LIN {X 18.5886,Y -15.8866,Z 59,A -46.5313,B 24.8302,C -3.0055,E1 25.1236,E2 -590.8316} C_DIS
LIN {X 19.6781,Y -14.5155,Z 59,A -42.6905,B 24.8293,C -3.0134,E1 25.1302,E2 -594.6728} C_DIS
LIN {X 20.6505,Y -13.0952,Z 59,A -38.2707,B 24.8276,C -3.0286,E1 25.1369,E2 -599.1068} C_DIS
LIN {X 21.5809,Y -11.4976,Z 59,A -33.8411,B 24.8261,C -3.042,E1 25.1429,E2 -603.5448} C_DIS
LIN {X 22.5618,Y -9.427,Z 59,A -28.8945,B 24.8248,C -3.053,E1 25.1486,E2 -608.4907} C_DIS
LIN {X 23.1997,Y -7.7258,Z 59,A -24.8284,B 24.8236,C -3.0637,E1 25.1524,E2 -612.5593} C_DIS
LIN {X 23.7063,Y -5.9947,Z 59,A -20.176,B 24.8215,C -3.0815,E1 25.1558,E2 -617.227} C_DIS
LIN {X 24.1573,Y -3.7876,Z 59,A -15.7991,B 24.8208,C -3.0876,E1 25.158,E2 -621.593} C_DIS
LIN {X 24.3666,Y -2.0474,Z 59,A -10.6689,B 24.8179,C -3.1121,E1 25.1595,E2 -626.7507} C_DIS
LIN {X 24.4517,Y -0.2551,Z 59,A -7.3543,B 24.8176,C -3.1151,E1 25.1598,E2 -630.0527} C_DIS
LIN {X 24.4235,Y 1.1938,Z 59,A -3.513,B 24.8157,C -3.1307,E1 25.1594,E2 -633.9081} C_DIS
LIN {X 24.2637,Y 3.0317,Z 59,A 0.5591,B 24.8145,C -3.1412,E1 25.1582,E2 -637.9809} C_DIS
LIN {X 24.0349,Y 4.4987,Z 59,A 3.954,B 24.8133,C -3.1508,E1 25.1566,E2 -641.3787} C_DIS
LIN {X 23.7384,Y 5.8651,Z 59,A 7.4962,B 24.8118,C -3.1636,E1 25.1543,E2 -644.9306} C_DIS
LIN {X 23.2116,Y 7.69,Z 59,A 11.9028,B 24.8103,C -3.176,E1 25.1507,E2 -649.3418} C_DIS
LIN {X 22.5143,Y 9.5408,Z 59,A 16.3866,B 24.8089,C -3.1874,E1 25.1461,E2 -653.8278} C_DIS
LIN {X 21.6112,Y 11.4401,Z 59,A 22.0841,B 24.8063,C -3.2091,E1 25.1389,E2 -659.5463} C_DIS
LIN {X 20.7577,Y 12.9244,Z 59,A 26.3239,B 24.8048,C -3.2218,E1 25.1326,E2 -663.7947} C_DIS
LIN {X 18.7966,Y 15.6399,Z 59,A 33.2506,B 24.8037,C -3.2304,E1 25.1209,E2 -670.7089} C_DIS
LIN {X 17.7343,Y 16.8352,Z 59,A 36.5534,B 24.8033,C -3.2339,E1 25.1146,E2 -674.0055} C_DIS
LIN {X 16.8552,Y 17.7155,Z 59,A 39.4969,B 24.8025,C -3.2401,E1 25.1087,E2 -676.9514} C_DIS
LIN {X 15.8547,Y 18.6158,Z 59,A 42.7481,B 24.8017,C -3.2471,E1 25.1019,E2 -680.2064} C_DIS
LIN {X 14.6509,Y 19.5773,Z 59,A 46.319,B 24.801,C -3.253,E1 25.094,E2 -683.7783} C_DIS
LIN {X 13.6252,Y 20.3048,Z 59,A 50.0535,B 24.7994,C -3.2654,E1 25.0853,E2 -687.5296} C_DIS
LIN {X 11.2373,Y 21.717,Z 59,A 55.8634,B 24.7992,C -3.2675,E1 25.0712,E2 -693.3275} C_DIS
LIN {X 9.712,Y 22.4407,Z 59,A 59.7569,B 24.7987,C -3.2713,E1 25.0613,E2 -697.2203} C_DIS
LIN {X 8.2716,Y 23.0108,Z 59,A 63.2886,B 24.7984,C -3.2738,E1 25.0521,E2 -700.7502} C_DIS
LIN {X 6.917,Y 23.4536,Z 59,A 66.6476,B 24.7981,C -3.2764,E1 25.0431,E2 -704.1094} C_DIS
LIN {X 5.5749,Y 23.8085,Z 59,A 70.5455,B 24.7971,C -3.2838,E1 25.0325,E2 -708.0193} C_DIS
LIN {X 2.8146,Y 24.2899,Z 59,A 77.442,B 24.7966,C -3.2882,E1 25.0135,E2 -714.9203} C_DIS
LIN {X -0.1109,Y 24.4522,Z 59,A 83.2288,B 24.7978,C -3.2789,E1 24.9974,E2 -720.6834} C_DIS
LIN {X -1.4173,Y 24.4113,Z 59,A 86.518,B 24.7977,C -3.2796,E1 24.9882,E2 -723.9752} C_DIS
LIN {X -3.0857,Y 24.257,Z 59,A 90.138,B 24.7982,C -3.2752,E1 24.9782,E2 -727.5869} C_DIS
LIN {X -4.2341,Y 24.0829,Z 59,A 92.9532,B 24.7984,C -3.274,E1 24.9704,E2 -730.4018} C_DIS
LIN {X -5.4753,Y 23.8315,Z 59,A 96.17,B 24.7984,C -3.2733,E1 24.9616,E2 -733.621} C_DIS
LIN {X -7.1047,Y 23.3973,Z 59,A 99.9316,B 24.7991,C -3.2679,E1 24.9516,E2 -737.3756} C_DIS
LIN {X -8.4462,Y 22.9473,Z 59,A 103.0268,B 24.7998,C -3.2624,E1 24.9434,E2 -740.4636} C_DIS
LIN {X -9.6923,Y 22.4495,Z 59,A 106.2631,B 24.8003,C -3.2587,E1 24.9351,E2 -743.6984} C_DIS
LIN {X -11.1641,Y 21.755,Z 59,A 110.5778,B 24.8006,C -3.2561,E1 24.9242,E2 -748.0182} C_DIS
LIN {X -12.5928,Y 20.9606,Z 59,A 114.1181,B 24.8016,C -3.2476,E1 24.9157,E2 -751.5488} C_DIS
LIN {X -13.6867,Y 20.2631,Z 59,A 117.0453,B 24.8024,C -3.2413,E1 24.9089,E2 -754.4703} C_DIS
LIN {X -14.7669,Y 19.4902,Z 59,A 120.374,B 24.803,C -3.2363,E1 24.9014,E2 -757.799} C_DIS
LIN {X -15.7348,Y 18.7176,Z 59,A 123.5618,B 24.8036,C -3.2318,E1 24.8946,E2 -760.9883} C_DIS
LIN {X -16.8114,Y 17.7567,Z 59,A 126.716,B 24.8046,C -3.2229,E1 24.8881,E2 -764.1338} C_DIS
LIN {X -17.8902,Y 16.6695,Z 59,A 130.2413,B 24.8057,C -3.214,E1 24.8813,E2 -767.653} C_DIS
LIN {X -18.8464,Y 15.58,Z 59,A 133.4231,B 24.8069,C -3.2043,E1 24.8755,E2 -770.8262} C_DIS
LIN {X -19.4761,Y 14.7856,Z 59,A 135.9661,B 24.8075,C -3.1991,E1 24.8712,E2 -773.3688} C_DIS
LIN {X -20.2128,Y 13.7609,Z 59,A 138.8623,B 24.8085,C -3.1909,E1 24.8666,E2 -776.2596} C_DIS
LIN {X -21.0039,Y 12.5205,Z 59,A 142.4582,B 24.8096,C -3.1822,E1 24.8613,E2 -779.853} C_DIS
LIN {X -21.8102,Y 11.0559,Z 59,A 146.4027,B 24.8109,C -3.1712,E1 24.8561,E2 -783.7921} C_DIS
LIN {X -22.4864,Y 9.6064,Z 59,A 150.4506,B 24.812,C -3.1618,E1 24.8515,E2 -787.8398} C_DIS
LIN {X -23.125,Y 7.9471,Z 59,A 154.1491,B 24.8138,C -3.147,E1 24.848,E2 -791.5236} C_DIS
LIN {X -23.7331,Y 5.8877,Z 59,A 160.6118,B 24.8147,C -3.1389,E1 24.8432,E2 -798.0045} C_DIS
LIN {X -24.2129,Y 3.4137,Z 59,A 165.9491,B 24.8173,C -3.1177,E1 24.8409,E2 -803.3226} C_DIS
LIN {X -24.4274,Y 1.1046,Z 59,A 171.0652,B 24.8194,C -3.0991,E1 24.8398,E2 -808.4249} C_DIS
LIN {X -24.4438,Y -0.648,Z 59,A 175.2842,B 24.8209,C -3.0869,E1 24.8399,E2 -812.6401} C_DIS
LIN {X -24.3255,Y -2.4847,Z 59,A 179.0868,B 24.8227,C -3.071,E1 24.8408,E2 -816.4276} C_DIS
LIN {X -24.2029,Y -3.4835,Z 59,A -178.0137,B 24.8232,C -3.0666,E1 24.8419,E2 -819.3337} C_DIS
LIN {X -23.8694,Y -5.3059,Z 59,A -173.6612,B 24.8247,C -3.0536,E1 24.8443,E2 -823.6807} C_DIS
LIN {X -23.394,Y -7.1158,Z 59,A -169.7271,B 24.8265,C -3.0383,E1 24.8472,E2 -827.6011} C_DIS
LIN {X -23.0263,Y -8.2283,Z 59,A -166.7651,B 24.8273,C -3.0315,E1 24.8499,E2 -830.5638} C_DIS
LIN {X -22.5113,Y -9.5477,Z 59,A -163.373,B 24.8283,C -3.0226,E1 24.8535,E2 -833.9535} C_DIS
LIN {X -21.682,Y -11.3053,Z 59,A -158.0978,B 24.8292,C -3.0143,E1 24.86,E2 -839.2372} C_DIS
LIN {X -20.7822,Y -12.8851,Z 59,A -154.6803,B 24.831,C -2.9987,E1 24.8649,E2 -842.6349} C_DIS
LIN {X -19.9758,Y -14.1032,Z 59,A -150.8673,B 24.8317,C -2.9925,E1 24.8709,E2 -846.4521} C_DIS
LIN {X -18.9459,Y -15.4589,Z 59,A -146.8113,B 24.8327,C -2.9837,E1 24.8779,E2 -850.506} C_DIS
LIN {X -18.0018,Y -16.5486,Z 59,A -143.8162,B 24.8338,C -2.974,E1 24.8835,E2 -853.4914} C_DIS
LIN {X -17.0433,Y -17.5344,Z 59,A -140.2269,B 24.8343,C -2.9697,E1 24.8906,E2 -857.0855} C_DIS
LIN {X -15.8934,Y -18.5828,Z 59,A -136.4143,B 24.8349,C -2.9639,E1 24.8986,E2 -860.8992} C_DIS
LIN {X -14.4257,Y -19.7434,Z 59,A -132.2434,B 24.8359,C -2.955,E1 24.9078,E2 -865.0639} C_DIS
LIN {X -13.0611,Y -20.6721,Z 59,A -128.5517,B 24.8367,C -2.9479,E1 24.9164,E2 -868.7508} C_DIS
LIN {X -11.9689,Y -21.3229,Z 59,A -125.2993,B 24.8369,C -2.9457,E1 24.9243,E2 -872.0076} C_DIS
LIN {X -10.5179,Y -22.0746,Z 59,A -121.576,B 24.8375,C -2.9404,E1 24.9336,E2 -875.7282} C_DIS
LIN {X -9.2022,Y -22.6548,Z 59,A -118.2938,B 24.838,C -2.9364,E1 24.942,E2 -879.0084} C_DIS
LIN {X -7.4566,Y -23.2877,Z 59,A -113.1727,B 24.8377,C -2.9387,E1 24.9556,E2 -884.1447} C_DIS
LIN {X -5.1579,Y -23.9018,Z 59,A -107.8107,B 24.8382,C -2.9342,E1 24.9702,E2 -889.5033} C_DIS
LIN {X -3.0281,Y -24.2644,Z 59,A -103.1173,B 24.8387,C -2.93,E1 24.9831,E2 -894.1907} C_DIS
LIN {X -1.3953,Y -24.4125,Z 59,A -99.4458,B 24.8388,C -2.9286,E1 24.9933,E2 -897.8603} C_DIS
LIN {X -0.0174,Y -24.4501,Z 59,A -95.7636,B 24.8383,C -2.9331,E1 25.0036,E2 -901.5533} C_DIS
Enddeposition()
LIN {X -0.0174,Y -24.4501,Z 59,A -95.7636,B 24.8383,C -2.9331,E1 25.0036,E2 -901.5533} C_DIS
Startdeposition()
$VEL.CP = VEL_PRINT
LIN {X -0.7566,Y -23.4595,Z 59,A -99.8079,B 24.8385,C -2.9315,E1 24.9923,E2 -897.5049} C_DIS
LIN {X -2.24,Y -23.3646,Z 59,A -103.1907,B 24.8383,C -2.9334,E1 24.9829,E2 -894.1253} C_DIS
LIN {X -4.0523,Y -23.119,Z 59,A -108.7197,B 24.839,C -2.9268,E1 24.9676,E2 -888.5755} C_DIS
LIN {X -6.4826,Y -22.5585,Z 59,A -114.2096,B 24.8382,C -2.9344,E1 24.9528,E2 -883.0957} C_DIS
LIN {X -8.3976,Y -21.918,Z 59,A -118.87,B 24.8375,C -2.9403,E1 24.9406,E2 -878.4403} C_DIS
LIN {X -9.7252,Y -21.3622,Z 59,A -122.3306,B 24.8371,C -2.9443,E1 24.9317,E2 -874.981} C_DIS
LIN {X -11.0217,Y -20.723,Z 59,A -126.0243,B 24.8367,C -2.9476,E1 24.9225,E2 -871.2851} C_DIS
LIN {X -12.3434,Y -19.9641,Z 59,A -130.4199,B 24.8367,C -2.9487,E1 24.912,E2 -866.8786} C_DIS
LIN {X -14.7063,Y -18.2932,Z 59,A -136.7323,B 24.8348,C -2.965,E1 24.8979,E2 -860.5828} C_DIS
LIN {X -16.2992,Y -16.8894,Z 59,A -142.4583,B 24.834,C -2.972,E1 24.8861,E2 -854.8504} C_DIS
LIN {X -17.6687,Y -15.451,Z 59,A -146.7467,B 24.8325,C -2.9855,E1 24.878,E2 -850.5753} C_DIS
LIN {X -18.4925,Y -14.4546,Z 59,A -150.2867,B 24.8319,C -2.9907,E1 24.8719,E2 -847.0311} C_DIS
LIN {X -19.7528,Y -12.6785,Z 59,A -156.7954,B 24.8311,C -2.9979,E1 24.8618,E2 -840.507} C_DIS
LIN {X -21.4854,Y -9.4496,Z 59,A -164.4593,B 24.8276,C -3.0281,E1 24.8523,E2 -832.8743} C_DIS
LIN {X -22.201,Y -7.6183,Z 59,A -169.7315,B 24.8263,C -3.0396,E1 24.8472,E2 -827.5998} C_DIS
LIN {X -22.6887,Y -6.0115,Z 59,A -173.3697,B 24.8247,C -3.0538,E1 24.8445,E2 -823.9744} C_DIS
LIN {X -23.0897,Y -4.2169,Z 59,A -178.0645,B 24.8232,C -3.0663,E1 24.8419,E2 -819.2821} C_DIS
LIN {X -23.3405,Y -2.4768,Z 59,A 177.6539,B 24.8217,C -3.0795,E1 24.8404,E2 -815.0064} C_DIS
LIN {X -23.4459,Y -1.0944,Z 59,A 174.6173,B 24.8203,C -3.0915,E1 24.8399,E2 -811.9803} C_DIS
LIN {X -23.4743,Y 0.0061,Z 59,A 171.6499,B 24.8195,C -3.0986,E1 24.8398,E2 -809.012} C_DIS
LIN {X -23.4421,Y 1.1727,Z 59,A 168.9595,B 24.8184,C -3.1082,E1 24.8401,E2 -806.3285} C_DIS
LIN {X -23.3347,Y 2.5282,Z 59,A 165.9238,B 24.817,C -3.1198,E1 24.8409,E2 -803.3024} C_DIS
LIN {X -23.2094,Y 3.4996,Z 59,A 163.3224,B 24.8162,C -3.1263,E1 24.8419,E2 -800.701} C_DIS
LIN {X -23.0087,Y 4.6383,Z 59,A 160.4784,B 24.8152,C -3.135,E1 24.8433,E2 -797.8609} C_DIS
LIN {X -22.6607,Y 6.1161,Z 59,A 156.1081,B 24.8142,C -3.1434,E1 24.8463,E2 -793.4852} C_DIS
LIN {X -22.0717,Y 7.9848,Z 59,A 151.3663,B 24.8125,C -3.1579,E1 24.8506,E2 -788.7513} C_DIS
LIN {X -21.3267,Y 9.8027,Z 59,A 146.6518,B 24.8107,C -3.1724,E1 24.8558,E2 -784.0454} C_DIS
LIN {X -20.6441,Y 11.1687,Z 59,A 143.2131,B 24.8093,C -3.1844,E1 24.8602,E2 -780.6171} C_DIS
LIN {X -19.9745,Y 12.3268,Z 59,A 139.3439,B 24.8086,C -3.1905,E1 24.8658,E2 -776.7427} C_DIS
LIN {X -18.7763,Y 14.0843,Z 59,A 134.5536,B 24.8067,C -3.2062,E1 24.8736,E2 -771.9666} C_DIS
LIN {X -17.7244,Y 15.3868,Z 59,A 130.4777,B 24.8054,C -3.2166,E1 24.8808,E2 -767.8967} C_DIS
LIN {X -16.6046,Y 16.5888,Z 59,A 126.3636,B 24.8043,C -3.2256,E1 24.8888,E2 -763.7864} C_DIS
LIN {X -15.4233,Y 17.6928,Z 59,A 122.3779,B 24.8033,C -3.2342,E1 24.8971,E2 -759.8053} C_DIS
LIN {X -14.0336,Y 18.8139,Z 59,A 118.6924,B 24.8017,C -3.2469,E1 24.9051,E2 -756.1366} C_DIS
LIN {X -12.9967,Y 19.5451,Z 59,A 114.6641,B 24.8017,C -3.2476,E1 24.9144,E2 -752.0965} C_DIS
LIN {X -11.2994,Y 20.5732,Z 59,A 110.378,B 24.8002,C -3.2592,E1 24.9247,E2 -747.8253} C_DIS
LIN {X -10.3559,Y 21.0633,Z 59,A 107.7414,B 24.7997,C -3.2631,E1 24.9313,E2 -745.1908} C_DIS
LIN {X -9.2262,Y 21.5824,Z 59,A 104.1959,B 24.7996,C -3.2643,E1 24.9404,E2 -741.6398} C_DIS
LIN {X -7.2866,Y 22.3119,Z 59,A 99.0405,B 24.7989,C -3.2698,E1 24.9539,E2 -736.4875} C_DIS
LIN {X -5.7896,Y 22.7464,Z 59,A 95.8762,B 24.7979,C -3.2778,E1 24.9624,E2 -733.3375} C_DIS
LIN {X -4.3954,Y 23.0563,Z 59,A 91.7105,B 24.7981,C -3.2761,E1 24.9738,E2 -729.1628} C_DIS
LIN {X -2.1805,Y 23.3701,Z 59,A 86.397,B 24.7976,C -3.2802,E1 24.9885,E2 -723.8555} C_DIS
LIN {X -0.2789,Y 23.47,Z 59,A 81.5846,B 24.7976,C -3.2804,E1 25.002,E2 -719.0427} C_DIS
LIN {X 1.9061,Y 23.3936,Z 59,A 76.718,B 24.7971,C -3.2841,E1 25.0155,E2 -714.1867} C_DIS
LIN {X 3.2653,Y 23.2434,Z 59,A 73.4862,B 24.7971,C -3.2842,E1 25.0245,E2 -710.9579} C_DIS
LIN {X 4.5996,Y 23.0167,Z 59,A 69.9381,B 24.7975,C -3.281,E1 25.0342,E2 -707.4061} C_DIS
LIN {X 6.1137,Y 22.6611,Z 59,A 66.1029,B 24.7978,C -3.2786,E1 25.0446,E2 -703.5707} C_DIS
LIN {X 7.9401,Y 22.0878,Z 59,A 61.0766,B 24.7986,C -3.2718,E1 25.0579,E2 -698.5382} C_DIS
LIN {X 9.74,Y 21.3553,Z 59,A 56.5513,B 24.799,C -3.2687,E1 25.0695,E2 -694.0163} C_DIS
LIN {X 11.4779,Y 20.4734,Z 59,A 52.0566,B 24.7995,C -3.2649,E1 25.0806,E2 -689.5253} C_DIS
LIN {X 12.9118,Y 19.601,Z 59,A 48.2651,B 24.7999,C -3.2616,E1 25.0895,E2 -685.7381} C_DIS
LIN {X 14.216,Y 18.6768,Z 59,A 44.1253,B 24.801,C -3.2528,E1 25.0989,E2 -681.5922} C_DIS
LIN {X 15.2415,Y 17.8498,Z 59,A 41.0755,B 24.8015,C -3.2485,E1 25.1054,E2 -678.5437} C_DIS
LIN {X 16.2351,Y 16.9512,Z 59,A 37.284,B 24.8029,C -3.237,E1 25.1132,E2 -674.7405} C_DIS
LIN {X 17.6696,Y 15.4499,Z 59,A 32.7149,B 24.8037,C -3.231,E1 25.1218,E2 -670.1772} C_DIS
LIN {X 18.7768,Y 14.0836,Z 59,A 27.8748,B 24.8055,C -3.2156,E1 25.1302,E2 -665.3232} C_DIS
LIN {X 19.7698,Y 12.652,Z 59,A 24.1734,B 24.8061,C -3.2106,E1 25.1359,E2 -661.6284} C_DIS
LIN {X 20.4022,Y 11.605,Z 59,A 21.341,B 24.8069,C -3.2044,E1 25.1399,E2 -658.796} C_DIS
LIN {X 20.9355,Y 10.6125,Z 59,A 18.606,B 24.8078,C -3.1972,E1 25.1434,E2 -656.0584} C_DIS
LIN {X 21.4846,Y 9.4514,Z 59,A 15.3153,B 24.809,C -3.187,E1 25.1472,E2 -652.7613} C_DIS
LIN {X 22.0181,Y 8.131,Z 59,A 11.9257,B 24.8101,C -3.1781,E1 25.1507,E2 -649.3693} C_DIS
LIN {X 22.5943,Y 6.3564,Z 59,A 6.6006,B 24.8126,C -3.1566,E1 25.155,E2 -644.0238} C_DIS
LIN {X 23.0799,Y 4.271,Z 59,A 1.5236,B 24.8143,C -3.1425,E1 25.1578,E2 -638.9429} C_DIS
LIN {X 23.3888,Y 1.972,Z 59,A -3.5176,B 24.8156,C -3.1317,E1 25.1594,E2 -633.906} C_DIS
LIN {X 23.4673,Y 0.4487,Z 59,A -7.1134,B 24.8168,C -3.1215,E1 25.1598,E2 -630.3074} C_DIS
LIN {X 23.4535,Y -0.9213,Z 59,A -10.8713,B 24.8185,C -3.1066,E1 25.1595,E2 -626.5366} C_DIS
LIN {X 23.2675,Y -3.0871,Z 59,A -15.1925,B 24.8192,C -3.1007,E1 25.1583,E2 -622.2269} C_DIS
LIN {X 23.0131,Y -4.617,Z 59,A -19.8726,B 24.8217,C -3.0793,E1 25.156,E2 -617.5236} C_DIS
LIN {X 22.4859,Y -6.7301,Z 59,A -24.9662,B 24.8234,C -3.0654,E1 25.1523,E2 -612.4262} C_DIS
LIN {X 22.0247,Y -8.1134,Z 59,A -28.197,B 24.8242,C -3.0582,E1 25.1493,E2 -609.1965} C_DIS
LIN {X 21.4205,Y -9.5954,Z 59,A -32.6846,B 24.8262,C -3.0405,E1 25.1443,E2 -604.6916} C_DIS
LIN {X 20.5634,Y -11.317,Z 59,A -37.0756,B 24.8274,C -3.0302,E1 25.1386,E2 -600.2994} C_DIS
LIN {X 19.6856,Y -12.783,Z 59,A -40.8219,B 24.8282,C -3.0231,E1 25.1331,E2 -596.5553} C_DIS
LIN {X 18.7709,Y -14.0915,Z 59,A -45.3793,B 24.8302,C -3.0059,E1 25.1256,E2 -591.9793} C_DIS
LIN {X 17.6664,Y -15.4536,Z 59,A -49.5654,B 24.8313,C -2.9961,E1 25.1181,E2 -587.7889} C_DIS
LIN {X 16.212,Y -16.9735,Z 59,A -53.8832,B 24.8317,C -2.9921,E1 25.1096,E2 -583.4801} C_DIS
LIN {X 15.3057,Y -17.7951,Z 59,A -57.1401,B 24.8328,C -2.9828,E1 25.1028,E2 -580.2139} C_DIS
LIN {X 14.1589,Y -18.7203,Z 59,A -61.1663,B 24.8341,C -2.971,E1 25.0939,E2 -576.1748} C_DIS
LIN {X 12.4,Y -19.9289,Z 59,A -66.595,B 24.8354,C -2.9591,E1 25.0812,E2 -570.7356} C_DIS
LIN {X 10.4354,Y -21.0242,Z 59,A -71.2033,B 24.8355,C -2.9581,E1 25.0699,E2 -566.1382} C_DIS
LIN {X 9.2637,Y -21.5662,Z 59,A -74.8919,B 24.8366,C -2.9486,E1 25.0604,E2 -562.436} C_DIS
LIN {X 7.5149,Y -22.236,Z 59,A -78.8963,B 24.8367,C -2.9478,E1 25.0499,E2 -558.438} C_DIS
LIN {X 5.6988,Y -22.7692,Z 59,A -84.2126,B 24.8379,C -2.9369,E1 25.0356,E2 -553.1045} C_DIS
LIN {X 4.305,Y -23.0732,Z 59,A -87.511,B 24.8381,C -2.9356,E1 25.0266,E2 -549.8068} C_DIS
LIN {X 2.5687,Y -23.3306,Z 59,A -91.2688,B 24.8379,C -2.9372,E1 25.0162,E2 -546.056} C_DIS
LIN {X 0.7947,Y -23.4581,Z 59,A -95.912,B 24.8383,C -2.933,E1 25.0032,E2 -541.4046} C_DIS
LIN {X 0.7947,Y -23.4581,Z 59,A -95.912,B 24.8383,C -2.933,E1 25.0032,E2 -541.4046} C_DIS
Enddeposition()
LIN {X 0.0063,Y -22.4836,Z 59,A -97.5185,B 24.8362,C -2.9523,E1 24.9989,E2 -539.8443} C_DIS
Startdeposition()
$VEL.CP = VEL_PRINT
LIN {X 1.5595,Y -22.4366,Z 59,A -92.0086,B 24.8347,C -2.9658,E1 25.0143,E2 -545.3846} C_DIS
LIN {X 3.1216,Y -22.2732,Z 59,A -88.1167,B 24.8345,C -2.9673,E1 25.0251,E2 -549.2772} C_DIS
LIN {X 4.708,Y -21.9925,Z 59,A -83.7759,B 24.8339,C -2.9726,E1 25.037,E2 -553.6256} C_DIS
LIN {X 6.4042,Y -21.5598,Z 59,A -79.6202,B 24.8337,C -2.9747,E1 25.0482,E2 -557.7794} C_DIS
LIN {X 7.3469,Y -21.2562,Z 59,A -76.7,B 24.833,C -2.9813,E1 25.0559,E2 -560.7095} C_DIS
LIN {X 9.2529,Y -20.4993,Z 59,A -72.0889,B 24.8327,C -2.9831,E1 25.0678,E2 -565.3143} C_DIS
LIN {X 10.257,Y -20.0158,Z 59,A -68.9742,B 24.832,C -2.9902,E1 25.0756,E2 -568.4373} C_DIS
LIN {X 11.5573,Y -19.2945,Z 59,A -64.9535,B 24.831,C -2.999,E1 25.0853,E2 -572.4669} C_DIS
LIN {X 13.2514,Y -18.1725,Z 59,A -59.8893,B 24.8299,C -3.0081,E1 25.097,E2 -577.5352} C_DIS
LIN {X 14.3458,Y -17.3216,Z 59,A -56.8684,B 24.8296,C -3.0107,E1 25.1035,E2 -580.5508} C_DIS
LIN {X 15.16,Y -16.6138,Z 59,A -54.186,B 24.829,C -3.0162,E1 25.1091,E2 -583.2356} C_DIS
LIN {X 16.2171,Y -15.5835,Z 59,A -49.4478,B 24.8269,C -3.0349,E1 25.1185,E2 -587.998} C_DIS
LIN {X 17.4501,Y -14.1892,Z 59,A -44.9108,B 24.8257,C -3.0448,E1 25.1266,E2 -592.5377} C_DIS
LIN {X 18.6917,Y -12.5087,Z 59,A -40.0505,B 24.8246,C -3.0543,E1 25.1344,E2 -597.3968} C_DIS
LIN {X 19.5379,Y -11.1403,Z 59,A -35.7673,B 24.8231,C -3.0677,E1 25.1405,E2 -601.6897} C_DIS
LIN {X 20.3402,Y -9.5976,Z 59,A -31.5687,B 24.8219,C -3.078,E1 25.1457,E2 -605.8904} C_DIS
LIN {X 20.8531,Y -8.4257,Z 59,A -28.233,B 24.8207,C -3.0885,E1 25.1493,E2 -609.2325} C_DIS
LIN {X 21.4888,Y -6.6387,Z 59,A -23.539,B 24.8191,C -3.1016,E1 25.1535,E2 -613.9312} C_DIS
LIN {X 21.8803,Y -5.205,Z 59,A -19.5859,B 24.8176,C -3.1151,E1 25.1562,E2 -617.8932} C_DIS
LIN {X 22.2269,Y -3.4358,Z 59,A -15.424,B 24.8164,C -3.1247,E1 25.1582,E2 -622.0537} C_DIS
LIN {X 22.3851,Y -2.1769,Z 59,A -12.3023,B 24.8154,C -3.1336,E1 25.1592,E2 -625.178} C_DIS
LIN {X 22.465,Y -1.0834,Z 59,A -9.1608,B 24.8139,C -3.1461,E1 25.1597,E2 -628.3304} C_DIS
LIN {X 22.4821,Y 0.6282,Z 59,A -5.1155,B 24.8127,C -3.1563,E1 25.1597,E2 -632.3758} C_DIS
LIN {X 22.4179,Y 1.8103,Z 59,A -1.4213,B 24.8107,C -3.1729,E1 25.1589,E2 -636.0874} C_DIS
LIN {X 22.0881,Y 4.2371,Z 59,A 4.4115,B 24.8089,C -3.1875,E1 25.1563,E2 -641.9206} C_DIS
LIN {X 21.8166,Y 5.4658,Z 59,A 7.7026,B 24.8077,C -3.198,E1 25.1541,E2 -645.2174} C_DIS
LIN {X 21.2687,Y 7.3134,Z 59,A 12.3729,B 24.8062,C -3.2097,E1 25.1502,E2 -649.8891} C_DIS
LIN {X 20.7199,Y 8.7478,Z 59,A 16.5733,B 24.8045,C -3.2237,E1 25.1457,E2 -654.0994} C_DIS
LIN {X 19.7745,Y 10.7145,Z 59,A 21.7076,B 24.8033,C -3.2343,E1 25.1393,E2 -659.2315} C_DIS
LIN {X 18.7691,Y 12.3919,Z 59,A 27.3347,B 24.8009,C -3.2534,E1 25.1309,E2 -664.8755} C_DIS
LIN {X 17.7328,Y 13.8346,Z 59,A 30.9233,B 24.8007,C -3.2548,E1 25.1249,E2 -668.4503} C_DIS
LIN {X 17.0052,Y 14.7197,Z 59,A 34.381,B 24.7993,C -3.2666,E1 25.1186,E2 -671.9203} C_DIS
LIN {X 16.1264,Y 15.6776,Z 59,A 37.4578,B 24.7987,C -3.2713,E1 25.1127,E2 -674.995} C_DIS
LIN {X 14.9896,Y 16.7675,Z 59,A 41.5848,B 24.7976,C -3.2803,E1 25.1042,E2 -679.1266} C_DIS
LIN {X 13.4278,Y 18.0425,Z 59,A 47.2925,B 24.7958,C -3.2946,E1 25.0916,E2 -684.8473} C_DIS
LIN {X 11.7259,Y 19.1918,Z 59,A 52.7579,B 24.7946,C -3.3045,E1 25.0786,E2 -690.3187} C_DIS
LIN {X 8.9904,Y 20.6157,Z 59,A 59.3358,B 24.7948,C -3.3027,E1 25.0622,E2 -696.8748} C_DIS
LIN {X 7.8987,Y 21.0583,Z 59,A 63.0509,B 24.7937,C -3.3115,E1 25.0525,E2 -700.6028} C_DIS
LIN {X 5.5842,Y 21.7866,Z 59,A 68.5908,B 24.7938,C -3.3105,E1 25.0377,E2 -706.1309} C_DIS
LIN {X 3.6103,Y 22.1989,Z 59,A 74.3953,B 24.7929,C -3.3177,E1 25.0217,E2 -711.9459} C_DIS
LIN {X 1.7287,Y 22.4243,Z 59,A 78.7212,B 24.7933,C -3.3144,E1 25.0097,E2 -716.2612} C_DIS
LIN {X 0.2984,Y 22.489,Z 59,A 82.7098,B 24.7931,C -3.3165,E1 24.9986,E2 -720.2541} C_DIS
LIN {X -1.7346,Y 22.4238,Z 59,A 87.8583,B 24.7933,C -3.3144,E1 24.9842,E2 -725.3991} C_DIS
LIN {X -3.1009,Y 22.2761,Z 59,A 90.9132,B 24.794,C -3.3093,E1 24.9758,E2 -728.4439} C_DIS
LIN {X -4.3996,Y 22.0562,Z 59,A 94.3468,B 24.7942,C -3.3073,E1 24.9664,E2 -731.8763} C_DIS
LIN {X -5.8627,Y 21.7132,Z 59,A 97.7933,B 24.795,C -3.3012,E1 24.9571,E2 -735.3132} C_DIS
LIN {X -7.1964,Y 21.3085,Z 59,A 102.1106,B 24.7949,C -3.302,E1 24.9456,E2 -739.6402} C_DIS
LIN {X -9.0507,Y 20.5893,Z 59,A 107.0424,B 24.7958,C -3.2943,E1 24.9329,E2 -744.5646} C_DIS
LIN {X -10.5621,Y 19.8567,Z 59,A 111.6425,B 24.7965,C -3.2893,E1 24.9214,E2 -749.1654} C_DIS
LIN {X -12.7433,Y 18.5326,Z 59,A 117.7721,B 24.7982,C -3.2753,E1 24.907,E2 -755.2811} C_DIS
LIN {X -14.1131,Y 17.5118,Z 59,A 122.1141,B 24.7993,C -3.2663,E1 24.8975,E2 -759.6174} C_DIS
LIN {X -15.494,Y 16.3021,Z 59,A 127.594,B 24.8001,C -3.26,E1 24.8862,E2 -765.1044} C_DIS
LIN {X -17.2694,Y 14.4086,Z 59,A 133.7435,B 24.8024,C -3.2414,E1 24.8748,E2 -771.2369} C_DIS
LIN {X -18.0982,Y 13.3529,Z 59,A 137.3465,B 24.8034,C -3.2334,E1 24.8688,E2 -774.838} C_DIS
LIN {X -19.3716,Y 11.427,Z 59,A 143.5201,B 24.8052,C -3.2186,E1 24.8597,E2 -781.0078} C_DIS
LIN {X -20.4415,Y 9.3802,Z 59,A 148.7887,B 24.8076,C -3.1989,E1 24.8532,E2 -786.2574} C_DIS
LIN {X -21.0891,Y 7.8158,Z 59,A 152.9207,B 24.8092,C -3.1852,E1 24.849,E2 -790.3799} C_DIS
LIN {X -21.5706,Y 6.3674,Z 59,A 157.107,B 24.8105,C -3.1748,E1 24.8455,E2 -794.5652} C_DIS
LIN {X -21.9946,Y 4.6981,Z 59,A 161.4909,B 24.8121,C -3.1613,E1 24.8427,E2 -798.9424} C_DIS
LIN {X -22.2215,Y 3.4701,Z 59,A 164.6539,B 24.8133,C -3.1513,E1 24.8413,E2 -802.1003} C_DIS
LIN {X -22.4059,Y 1.9516,Z 59,A 168.6053,B 24.8147,C -3.1394,E1 24.8402,E2 -806.0469} C_DIS
LIN {X -22.491,Y 0.1916,Z 59,A 173.2596,B 24.8162,C -3.1261,E1 24.8398,E2 -810.6974} C_DIS
LIN {X -22.4422,Y -1.4798,Z 59,A 177.3543,B 24.8179,C -3.1122,E1 24.8403,E2 -814.7834} C_DIS
LIN {X -22.2744,Y -3.1132,Z 59,A -178.9562,B 24.8196,C -3.0973,E1 24.8415,E2 -818.4592} C_DIS
LIN {X -22.0834,Y -4.2615,Z 59,A -175.442,B 24.8204,C -3.0907,E1 24.8432,E2 -821.9785} C_DIS
LIN {X -21.7202,Y -5.8371,Z 59,A -170.935,B 24.8216,C -3.0802,E1 24.8463,E2 -826.4868} C_DIS
LIN {X -21.0712,Y -7.8625,Z 59,A -165.6764,B 24.8235,C -3.0639,E1 24.8511,E2 -831.7362} C_DIS
LIN {X -20.4668,Y -9.324,Z 59,A -162.0416,B 24.825,C -3.0509,E1 24.8551,E2 -835.3599} C_DIS
LIN {X -19.6795,Y -10.8886,Z 59,A -156.7029,B 24.8259,C -3.0433,E1 24.8621,E2 -840.7089} C_DIS
LIN {X -18.7474,Y -12.4248,Z 59,A -152.8094,B 24.8276,C -3.0284,E1 24.8679,E2 -844.5864} C_DIS
LIN {X -17.9758,Y -13.517,Z 59,A -149.2375,B 24.8284,C -3.0211,E1 24.8738,E2 -848.1581} C_DIS
LIN {X -16.9692,Y -14.7609,Z 59,A -145.4445,B 24.8297,C -3.0105,E1 24.8806,E2 -851.9431} C_DIS
LIN {X -15.8356,Y -15.9711,Z 59,A -140.4248,B 24.8302,C -3.006,E1 24.8903,E2 -856.9737} C_DIS
LIN {X -14.4917,Y -17.2,Z 59,A -136.1429,B 24.8314,C -2.9953,E1 24.8993,E2 -861.2468} C_DIS
LIN {X -12.7625,Y -18.5192,Z 59,A -129.9358,B 24.832,C -2.9901,E1 24.9134,E2 -867.4632} C_DIS
LIN {X -10.8343,Y -19.7097,Z 59,A -124.3308,B 24.833,C -2.9812,E1 24.9269,E2 -873.0635} C_DIS
LIN {X -8.4755,Y -20.8327,Z 59,A -118.255,B 24.8342,C -2.9702,E1 24.9424,E2 -879.128} C_DIS
LIN {X -6.6301,Y -21.4913,Z 59,A -112.7306,B 24.8342,C -2.97,E1 24.957,E2 -884.6621} C_DIS
LIN {X -5.0369,Y -21.9196,Z 59,A -109.2702,B 24.8351,C -2.9625,E1 24.9664,E2 -888.1097} C_DIS
LIN {X -3.6205,Y -22.1977,Z 59,A -105.1026,B 24.8348,C -2.9649,E1 24.9778,E2 -892.2871} C_DIS
LIN {X -1.7681,Y -22.4211,Z 59,A -100.324,B 24.8348,C -2.9647,E1 24.9911,E2 -897.0678} C_DIS
LIN {X 0.0063,Y -22.4836,Z 59,A -97.5184,B 24.8362,C -2.9523,E1 24.9989,E2 -899.8443} C_DIS
Enddeposition()
LIN {X 0.0063,Y -22.4836,Z 59,A -97.5184,B 24.8362,C -2.9523,E1 24.9989,E2 -899.8443} C_DIS
Startdeposition()
$VEL.CP = VEL_PRINT
LIN {X -0.4377,Y -21.5055,Z 59,A -99.2003,B 24.8347,C -2.9656,E1 24.9943,E2 -898.1938} C_DIS
LIN {X -2.2395,Y -21.3932,Z 59,A -104.2253,B 24.8349,C -2.9642,E1 24.9803,E2 -893.1634} C_DIS
LIN {X -3.6879,Y -21.1918,Z 59,A -108.0465,B 24.8347,C -2.9657,E1 24.9697,E2 -889.3423} C_DIS
LIN {X -5.3273,Y -20.84,Z 59,A -112.2327,B 24.8343,C -2.9697,E1 24.9583,E2 -885.1601} C_DIS
LIN {X -6.6002,Y -20.4721,Z 59,A -115.5235,B 24.8338,C -2.9736,E1 24.9496,E2 -881.8731} C_DIS
LIN {X -7.7991,Y -20.0465,Z 59,A -119.777,B 24.8341,C -2.9714,E1 24.9384,E2 -877.6053} C_DIS
LIN {X -9.5193,Y -19.2885,Z 59,A -124.074,B 24.833,C -2.9811,E1 24.9276,E2 -873.3208} C_DIS
LIN {X -10.9024,Y -18.5425,Z 59,A -128.2851,B 24.8324,C -2.9864,E1 24.9173,E2 -869.1103} C_DIS
LIN {X -11.7438,Y -18.0206,Z 59,A -131.8074,B 24.8324,C -2.9856,E1 24.909,E2 -865.5747} C_DIS
LIN {X -13.7903,Y -16.5081,Z 59,A -137.9148,B 24.8307,C -3.0008,E1 24.8955,E2 -859.4813} C_DIS
LIN {X -14.8422,Y -15.5692,Z 59,A -141.6816,B 24.8299,C -3.0081,E1 24.8878,E2 -855.7166} C_DIS
LIN {X -15.6857,Y -14.7188,Z 59,A -145.1213,B 24.8293,C -3.0136,E1 24.8812,E2 -852.2751} C_DIS
LIN {X -16.7827,Y -13.4546,Z 59,A -148.9181,B 24.8278,C -3.0267,E1 24.8744,E2 -848.4922} C_DIS
LIN {X -17.7454,Y -12.1558,Z 59,A -154.2133,B 24.8271,C -3.0325,E1 24.8657,E2 -843.1852} C_DIS
LIN {X -19.0257,Y -10.0339,Z 59,A -161.5598,B 24.8255,C -3.0466,E1 24.8557,E2 -835.834} C_DIS
LIN {X -19.981,Y -7.9654,Z 59,A -167.2575,B 24.8234,C -3.065,E1 24.8495,E2 -830.1487} C_DIS
LIN {X -20.7514,Y -5.6627,Z 59,A -172.8559,B 24.8208,C -3.0873,E1 24.8449,E2 -824.5715} C_DIS
LIN {X -21.0992,Y -4.1852,Z 59,A -177.2735,B 24.8196,C -3.0979,E1 24.8423,E2 -820.1534} C_DIS
LIN {X -21.3085,Y -2.9393,Z 59,A 179.7428,B 24.8182,C -3.1096,E1 24.841,E2 -817.18} C_DIS
LIN {X -21.4305,Y -1.8507,Z 59,A 176.2503,B 24.8174,C -3.1164,E1 24.8401,E2 -813.6828} C_DIS
LIN {X -21.5115,Y 0.1039,Z 59,A 170.3691,B 24.8158,C -3.1301,E1 24.8399,E2 -807.799} C_DIS
LIN {X -21.3536,Y 2.5881,Z 59,A 164.9039,B 24.8128,C -3.1551,E1 24.8412,E2 -802.361} C_DIS
LIN {X -21.1869,Y 3.7155,Z 59,A 161.3732,B 24.8119,C -3.1627,E1 24.8428,E2 -798.8273} C_DIS
LIN {X -20.7418,Y 5.6975,Z 59,A 156.2688,B 24.8098,C -3.1805,E1 24.8461,E2 -793.7357} C_DIS
LIN {X -20.4134,Y 6.7804,Z 59,A 152.8419,B 24.8089,C -3.188,E1 24.8491,E2 -790.3072} C_DIS
LIN {X -19.8301,Y 8.3336,Z 59,A 148.7096,B 24.8072,C -3.2022,E1 24.8533,E2 -786.1859} C_DIS
LIN {X -19.1749,Y 9.7471,Z 59,A 144.2196,B 24.8059,C -3.2128,E1 24.8588,E2 -781.697} C_DIS
LIN {X -18.5111,Y 10.9554,Z 59,A 141.0448,B 24.8044,C -3.2251,E1 24.8632,E2 -778.5351} C_DIS
LIN {X -17.8688,Y 11.9747,Z 59,A 137.3508,B 24.8036,C -3.2318,E1 24.8688,E2 -774.8385} C_DIS
LIN {X -16.7637,Y 13.4784,Z 59,A 132.2949,B 24.802,C -3.2443,E1 24.8774,E2 -769.7885} C_DIS
LIN {X -15.7946,Y 14.6021,Z 59,A 128.5464,B 24.8007,C -3.2549,E1 24.8844,E2 -766.0486} C_DIS
LIN {X -15.0402,Y 15.378,Z 59,A 125.6301,B 24.7999,C -3.2614,E1 24.8901,E2 -763.1357} C_DIS
LIN {X -14.0113,Y 16.321,Z 59,A 122.1478,B 24.7988,C -3.2707,E1 24.8974,E2 -759.6619} C_DIS
LIN {X -13.1043,Y 17.0576,Z 59,A 118.9794,B 24.798,C -3.277,E1 24.9043,E2 -756.4966} C_DIS
LIN {X -12.0252,Y 17.8347,Z 59,A 115.5238,B 24.7971,C -3.2843,E1 24.9122,E2 -753.0466} C_DIS
LIN {X -11.211,Y 18.357,Z 59,A 112.5757,B 24.7967,C -3.287,E1 24.9192,E2 -750.0959} C_DIS
LIN {X -9.8216,Y 19.1369,Z 59,A 108.6493,B 24.7957,C -3.2957,E1 24.9288,E2 -746.1791} C_DIS
LIN {X -8.8748,Y 19.594,Z 59,A 105.4184,B 24.7954,C -3.2975,E1 24.937,E2 -742.9445} C_DIS
LIN {X -7.3564,Y 20.213,Z 59,A 101.0881,B 24.7947,C -3.3034,E1 24.9483,E2 -738.6191} C_DIS
LIN {X -5.7453,Y 20.7285,Z 59,A 96.5478,B 24.7941,C -3.3081,E1 24.9604,E2 -734.0822} C_DIS
LIN {X -4.0583,Y 21.1237,Z 59,A 91.9162,B 24.7937,C -3.3118,E1 24.973,E2 -729.454} C_DIS
LIN {X -2.9203,Y 21.3112,Z 59,A 88.9551,B 24.7933,C -3.3145,E1 24.9812,E2 -726.4968} C_DIS
LIN {X -1.455,Y 21.4607,Z 59,A 84.9064,B 24.7932,C -3.3155,E1 24.9925,E2 -722.4485} C_DIS
LIN {X -0.003,Y 21.5102,Z 59,A 80.6647,B 24.7934,C -3.3139,E1 25.0043,E2 -718.2029} C_DIS
LIN {X 2.2383,Y 21.3933,Z 59,A 75.4514,B 24.7928,C -3.319,E1 25.0188,E2 -713.0043} C_DIS
LIN {X 3.612,Y 21.2048,Z 59,A 71.2957,B 24.7933,C -3.3147,E1 25.0303,E2 -708.8421} C_DIS
LIN {X 5.0107,Y 20.9185,Z 59,A 67.7508,B 24.7933,C -3.3147,E1 25.0399,E2 -705.3021} C_DIS
LIN {X 6.2369,Y 20.5855,Z 59,A 64.3301,B 24.7936,C -3.3121,E1 25.0491,E2 -701.8811} C_DIS
LIN {X 7.7174,Y 20.0781,Z 59,A 60.3574,B 24.7939,C -3.31,E1 25.0595,E2 -697.9115} C_DIS
LIN {X 9.4411,Y 19.3274,Z 59,A 54.4876,B 24.7954,C -3.2975,E1 25.0744,E2 -692.0268} C_DIS
LIN {X 10.9568,Y 18.5101,Z 59,A 50.4555,B 24.7957,C -3.2958,E1 25.0842,E2 -688.0026} C_DIS
LIN {X 11.9829,Y 17.8633,Z 59,A 46.7984,B 24.7967,C -3.2872,E1 25.0927,E2 -684.3371} C_DIS
LIN {X 13.8023,Y 16.498,Z 59,A 41.447,B 24.7973,C -3.2826,E1 25.1045,E2 -678.9948} C_DIS
LIN {X 14.73,Y 15.6752,Z 59,A 38.3169,B 24.7979,C -3.2777,E1 25.1109,E2 -675.8657} C_DIS
LIN {X 15.8039,Y 14.5915,Z 59,A 33.2763,B 24.8001,C -3.2603,E1 25.1207,E2 -670.8056} C_DIS
LIN {X 16.8448,Y 13.3768,Z 59,A 28.464,B 24.8019,C -3.2454,E1 25.1291,E2 -665.9805} C_DIS
LIN {X 18.6886,Y 10.65,Z 59,A 21.3171,B 24.8027,C -3.2387,E1 25.1398,E2 -658.8535} C_DIS
LIN {X 19.177,Y 9.743,Z 59,A 17.8176,B 24.8045,C -3.2241,E1 25.1443,E2 -655.3379} C_DIS
LIN {X 20.1629,Y 7.4925,Z 59,A 11.6082,B 24.8063,C -3.209,E1 25.1509,E2 -649.127} C_DIS
LIN {X 20.7873,Y 5.5289,Z 59,A 5.8591,B 24.8086,C -3.1904,E1 25.1554,E2 -643.3666} C_DIS
LIN {X 21.1471,Y 3.9361,Z 59,A 2.2426,B 24.8093,C -3.1846,E1 25.1574,E2 -639.7574} C_DIS
LIN {X 21.3599,Y 2.5381,Z 59,A -1.9336,B 24.8112,C -3.169,E1 25.159,E2 -635.5689} C_DIS
LIN {X 21.4949,Y 0.808,Z 59,A -6.4895,B 24.8128,C -3.1553,E1 25.1597,E2 -631.0077} C_DIS
LIN {X 21.4736,Y -1.2525,Z 59,A -12.2398,B 24.8151,C -3.1356,E1 25.1592,E2 -625.2447} C_DIS
LIN {X 21.2617,Y -3.2599,Z 59,A -16.8958,B 24.8163,C -3.1261,E1 25.1576,E2 -620.5938} C_DIS
LIN {X 21.063,Y -4.3619,Z 59,A -20.7777,B 24.8184,C -3.1078,E1 25.1555,E2 -616.6912} C_DIS
LIN {X 20.3289,Y -7.0302,Z 59,A -26.9543,B 24.8196,C -3.0973,E1 25.1506,E2 -610.525} C_DIS
LIN {X 19.7226,Y -8.5844,Z 59,A -32.2632,B 24.8222,C -3.0755,E1 25.1449,E2 -605.1938} C_DIS
LIN {X 18.916,Y -10.2405,Z 59,A -36.8077,B 24.8234,C -3.065,E1 25.1391,E2 -600.6484} C_DIS
LIN {X 17.9845,Y -11.8,Z 59,A -41.3849,B 24.8247,C -3.0542,E1 25.1324,E2 -596.0687} C_DIS
LIN {X 17.2316,Y -12.8744,Z 59,A -44.7595,B 24.8256,C -3.046,E1 25.1269,E2 -592.6912} C_DIS
LIN {X 16.4957,Y -13.8052,Z 59,A -47.8307,B 24.8264,C -3.0388,E1 25.1215,E2 -589.6171} C_DIS
LIN {X 15.819,Y -14.5753,Z 59,A -50.767,B 24.8274,C -3.0301,E1 25.1159,E2 -586.6733} C_DIS
LIN {X 14.815,Y -15.5953,Z 59,A -54.5966,B 24.8285,C -3.021,E1 25.1083,E2 -582.8381} C_DIS
LIN {X 13.7703,Y -16.5246,Z 59,A -58.1149,B 24.8292,C -3.0147,E1 25.1009,E2 -579.3187} C_DIS
LIN {X 12.933,Y -17.1878,Z 59,A -61.0304,B 24.8299,C -3.0081,E1 25.0944,E2 -576.3983} C_DIS
LIN {X 11.8566,Y -17.947,Z 59,A -64.4261,B 24.8306,C -3.0023,E1 25.0866,E2 -573.0003} C_DIS
LIN {X 10.8281,Y -18.5863,Z 59,A -68.0332,B 24.8316,C -2.9932,E1 25.0779,E2 -569.3826} C_DIS
LIN {X 9.2674,Y -19.4113,Z 59,A -72.6855,B 24.8324,C -2.9861,E1 25.0663,E2 -564.726} C_DIS
LIN {X 7.8482,Y -20.0272,Z 59,A -76.7241,B 24.833,C -2.981,E1 25.0559,E2 -560.6847} C_DIS
LIN {X 6.2273,Y -20.5889,Z 59,A -81.3279,B 24.8336,C -2.9753,E1 25.0436,E2 -556.0761} C_DIS
LIN {X 5.0796,Y -20.9014,Z 59,A -84.8045,B 24.8342,C -2.9698,E1 25.0342,E2 -552.5915} C_DIS
LIN {X 2.9488,Y -21.3067,Z 59,A -90.1326,B 24.8343,C -2.969,E1 25.0195,E2 -547.267} C_DIS
LIN {X 1.5826,Y -21.4519,Z 59,A -93.6608,B 24.8344,C -2.9681,E1 25.0097,E2 -543.7388} C_DIS
LIN {X 0.0132,Y -21.5087,Z 59,A -97.4445,B 24.8343,C -2.9698,E1 24.9992,E2 -539.9598} C_DIS
Enddeposition()
LIN {X 0.0132,Y -21.5087,Z 59,A -97.4445,B 24.8343,C -2.9698,E1 24.9992,E2 -539.9598} C_DIS
Startdeposition()
$VEL.CP = VEL_PRINT
LIN {X 0.8872,Y -20.5099,Z 59,A -93.0523,B 24.8307,C -3.0017,E1 25.0116,E2 -544.4269} C_DIS
LIN {X 3.6268,Y -20.2064,Z 59,A -84.9087,B 24.8297,C -3.0102,E1 25.0342,E2 -552.5836} C_DIS
LIN {X 5.6471,Y -19.7375,Z 59,A -80.5568,B 24.8303,C -3.0046,E1 25.0459,E2 -556.9155} C_DIS
LIN {X 6.6026,Y -19.4386,Z 59,A -77.5592,B 24.8298,C -3.0095,E1 25.0539,E2 -559.9192} C_DIS
LIN {X 7.9955,Y -18.9084,Z 59,A -73.4239,B 24.8291,C -3.015,E1 25.0646,E2 -564.0582} C_DIS
LIN {X 8.9802,Y -18.4609,Z 59,A -70.562,B 24.8288,C -3.0183,E1 25.0718,E2 -566.9206} C_DIS
LIN {X 10.0962,Y -17.8754,Z 59,A -67.1804,B 24.8282,C -3.023,E1 25.0802,E2 -570.3038} C_DIS
LIN {X 11.393,Y -17.0774,Z 59,A -62.1216,B 24.8265,C -3.0381,E1 25.0921,E2 -575.3819} C_DIS
LIN {X 12.8343,Y -16.0224,Z 59,A -56.9634,B 24.8251,C -3.05,E1 25.1035,E2 -580.5495} C_DIS
LIN {X 14.1163,Y -14.906,Z 59,A -52.7332,B 24.8244,C -3.056,E1 25.1122,E2 -584.7768} C_DIS
LIN {X 15.2752,Y -13.7157,Z 59,A -48.0752,B 24.8231,C -3.0675,E1 25.1211,E2 -589.4416} C_DIS
LIN {X 16.3818,Y -12.3727,Z 59,A -42.8887,B 24.8213,C -3.0832,E1 25.1301,E2 -594.641} C_DIS
LIN {X 17.4692,Y -10.784,Z 59,A -37.767,B 24.8199,C -3.0954,E1 25.1379,E2 -599.7661} C_DIS
LIN {X 18.4331,Y -9.0373,Z 59,A -33.168,B 24.8191,C -3.1019,E1 25.1439,E2 -604.3562} C_DIS
LIN {X 18.9387,Y -7.9232,Z 59,A -28.7579,B 24.8168,C -3.1217,E1 25.1489,E2 -608.7893} C_DIS
LIN {X 19.5262,Y -6.3385,Z 59,A -24.1861,B 24.8153,C -3.1345,E1 25.153,E2 -613.3656} C_DIS
LIN {X 19.9887,Y -4.6803,Z 59,A -19.851,B 24.8141,C -3.1445,E1 25.1561,E2 -617.6995} C_DIS
LIN {X 20.2287,Y -3.5014,Z 59,A -16.1358,B 24.8124,C -3.1585,E1 25.158,E2 -621.4262} C_DIS
LIN {X 20.3985,Y -2.3131,Z 59,A -13.1161,B 24.8115,C -3.1657,E1 25.159,E2 -624.445} C_DIS
LIN {X 20.5017,Y -1.0663,Z 59,A -9.4033,B 24.81,C -3.1788,E1 25.1597,E2 -628.1668} C_DIS
LIN {X 20.5264,Y 0.3459,Z 59,A -5.3704,B 24.8084,C -3.192,E1 25.1597,E2 -632.207} C_DIS
LIN {X 20.4264,Y 2.0537,Z 59,A -1.1101,B 24.8072,C -3.2016,E1 25.1588,E2 -636.4647} C_DIS
LIN {X 20.2422,Y 3.422,Z 59,A 3.165,B 24.8053,C -3.2175,E1 25.1569,E2 -640.7525} C_DIS
LIN {X 19.9382,Y 4.8911,Z 59,A 7.1105,B 24.8041,C -3.2277,E1 25.1545,E2 -644.699} C_DIS
LIN {X 19.6286,Y 6.0141,Z 59,A 10.4107,B 24.8028,C -3.2377,E1 25.1519,E2 -648.0041} C_DIS
LIN {X 19.0729,Y 7.5943,Z 59,A 14.8928,B 24.8014,C -3.2491,E1 25.1475,E2 -652.4883} C_DIS
LIN {X 18.5381,Y 8.8198,Z 59,A 19.1502,B 24.7996,C -3.2644,E1 25.1425,E2 -656.7589} C_DIS
LIN {X 17.5488,Y 10.6533,Z 59,A 24.5192,B 24.7982,C -3.2753,E1 25.1351,E2 -662.1259} C_DIS
LIN {X 16.6353,Y 12.0299,Z 59,A 29.538,B 24.7963,C -3.2903,E1 25.1271,E2 -667.1559} C_DIS
LIN {X 15.6617,Y 13.2728,Z 59,A 33.1944,B 24.7959,C -3.2936,E1 25.1207,E2 -670.803} C_DIS
LIN {X 15.0079,Y 14.007,Z 59,A 36.0513,B 24.7951,C -3.3005,E1 25.1153,E2 -673.6638} C_DIS
LIN {X 13.8464,Y 15.157,Z 59,A 40.7348,B 24.7938,C -3.3107,E1 25.1058,E2 -678.3522} C_DIS
LIN {X 12.755,Y 16.0861,Z 59,A 44.5974,B 24.793,C -3.3168,E1 25.0975,E2 -682.2146} C_DIS
LIN {X 11.8181,Y 16.7867,Z 59,A 47.7988,B 24.7924,C -3.3217,E1 25.0903,E2 -685.4163} C_DIS
LIN {X 10.7635,Y 17.4817,Z 59,A 52.8704,B 24.7901,C -3.3398,E1 25.0782,E2 -690.5149} C_DIS
LIN {X 7.5201,Y 19.1024,Z 59,A 62.719,B 24.789,C -3.3487,E1 25.0531,E2 -700.3601} C_DIS
LIN {X 4.832,Y 19.9526,Z 59,A 69.285,B 24.7896,C -3.3442,E1 25.0356,E2 -706.9042} C_DIS
LIN {X 3.6254,Y 20.2064,Z 59,A 73.0286,B 24.7891,C -3.3477,E1 25.0253,E2 -710.6519} C_DIS
LIN {X 2.0574,Y 20.4261,Z 59,A 77.9588,B 24.7886,C -3.352,E1 25.0116,E2 -715.5888} C_DIS
LIN {X -0.5799,Y 20.5212,Z 59,A 84.5244,B 24.7894,C -3.3456,E1 24.9933,E2 -722.1382} C_DIS
LIN {X -1.6153,Y 20.4656,Z 59,A 87.3952,B 24.7896,C -3.3442,E1 24.9853,E2 -725.0069} C_DIS
LIN {X -2.7474,Y 20.3448,Z 59,A 90.9853,B 24.7895,C -3.345,E1 24.9754,E2 -728.6013} C_DIS
LIN {X -4.3564,Y 20.0614,Z 59,A 94.8558,B 24.7904,C -3.3373,E1 24.9648,E2 -732.4577} C_DIS
LIN {X -5.6125,Y 19.7471,Z 59,A 99.6012,B 24.7901,C -3.3402,E1 24.952,E2 -737.2174} C_DIS
LIN {X -7.312,Y 19.1829,Z 59,A 103.9904,B 24.7913,C -3.3307,E1 24.9405,E2 -741.5925} C_DIS
LIN {X -8.8808,Y 18.509,Z 59,A 109.0264,B 24.792,C -3.3252,E1 24.9277,E2 -746.6277} C_DIS
LIN {X -10.5368,Y 17.6189,Z 59,A 114.2799,B 24.7931,C -3.3163,E1 24.9149,E2 -751.8753} C_DIS
LIN {X -11.8292,Y 16.7785,Z 59,A 118.6353,B 24.7941,C -3.3083,E1 24.9049,E2 -756.2263} C_DIS
LIN {X -13.3049,Y 15.6344,Z 59,A 124.0144,B 24.7954,C -3.2981,E1 24.8933,E2 -761.6011} C_DIS
LIN {X -14.6946,Y 14.3361,Z 59,A 128.7271,B 24.7972,C -3.2832,E1 24.8839,E2 -766.2978} C_DIS
LIN {X -15.5404,Y 13.415,Z 59,A 132.4375,B 24.7982,C -3.2755,E1 24.877,E2 -770.0066} C_DIS
LIN {X -16.2965,Y 12.4852,Z 59,A 135.9573,B 24.7991,C -3.2677,E1 24.8709,E2 -773.5243} C_DIS
LIN {X -17.1921,Y 11.2202,Z 59,A 139.8431,B 24.8008,C -3.2543,E1 24.8648,E2 -777.3972} C_DIS
LIN {X -17.7619,Y 10.2944,Z 59,A 142.9741,B 24.8018,C -3.2463,E1 24.8604,E2 -780.5252} C_DIS
LIN {X -18.3586,Y 9.1881,Z 59,A 146.7497,B 24.8029,C -3.2373,E1 24.8555,E2 -784.2995} C_DIS
LIN {X -18.8998,Y 8.0158,Z 59,A 150.1812,B 24.8042,C -3.2261,E1 24.8516,E2 -787.723} C_DIS
LIN {X -19.3252,Y 6.9274,Z 59,A 153.4961,B 24.8054,C -3.2166,E1 24.8484,E2 -791.0338} C_DIS
LIN {X -19.7704,Y 5.5304,Z 59,A 157.8952,B 24.8068,C -3.2053,E1 24.8449,E2 -795.4313} C_DIS
LIN {X -20.112,Y 4.1184,Z 59,A 161.6554,B 24.8084,C -3.1918,E1 24.8426,E2 -799.181} C_DIS
LIN {X -20.355,Y 2.6696,Z 59,A 166.6194,B 24.8096,C -3.1822,E1 24.8406,E2 -804.1518} C_DIS
LIN {X -20.5193,Y 0.6425,Z 59,A 171.3336,B 24.8121,C -3.161,E1 24.8398,E2 -808.8434} C_DIS
LIN {X -20.524,Y -0.4681,Z 59,A 174.7259,B 24.8131,C -3.1524,E1 24.8398,E2 -812.2356} C_DIS
LIN {X -20.4556,Y -1.7376,Z 59,A 178.6299,B 24.8143,C -3.1428,E1 24.8407,E2 -816.14} C_DIS
LIN {X -20.254,Y -3.3514,Z 59,A -176.9929,B 24.816,C -3.1284,E1 24.8424,E2 -820.5087} C_DIS
LIN {X -20.0244,Y -4.5246,Z 59,A -173.961,B 24.8173,C -3.1172,E1 24.8442,E2 -823.5317} C_DIS
LIN {X -19.7821,Y -5.4881,Z 59,A -170.6334,B 24.818,C -3.1112,E1 24.8466,E2 -826.8642} C_DIS
LIN {X -19.2197,Y -7.2144,Z 59,A -165.7459,B 24.8198,C -3.0959,E1 24.8511,E2 -831.743} C_DIS
LIN {X -18.7426,Y -8.3764,Z 59,A -162.5681,B 24.8211,C -3.0849,E1 24.8546,E2 -834.9119} C_DIS
LIN {X -18.0738,Y -9.7358,Z 59,A -157.7315,B 24.8221,C -3.0761,E1 24.8608,E2 -839.7534} C_DIS
LIN {X -16.7845,Y -11.8198,Z 59,A -149.5379,B 24.8234,C -3.0653,E1 24.8734,E2 -847.9619} C_DIS
LIN {X -15.4872,Y -13.4758,Z 59,A -144.5139,B 24.8253,C -3.0481,E1 24.8825,E2 -852.9679} C_DIS
LIN {X -13.9548,Y -15.057,Z 59,A -139.1997,B 24.8272,C -3.0316,E1 24.893,E2 -858.265} C_DIS
LIN {X -13.0887,Y -15.8159,Z 59,A -134.8248,B 24.8272,C -3.0316,E1 24.9024,E2 -862.6567} C_DIS
LIN {X -10.6845,Y -17.5298,Z 59,A -127.6921,B 24.8294,C -3.0129,E1 24.9189,E2 -869.7683} C_DIS
LIN {X -8.961,Y -18.4701,Z 59,A -121.3044,B 24.8296,C -3.0113,E1 24.9347,E2 -876.1696} C_DIS
LIN {X -7.33,Y -19.1762,Z 59,A -117.2254,B 24.8307,C -3.0013,E1 24.9452,E2 -880.2338} C_DIS
LIN {X -5.9787,Y -19.6394,Z 59,A -112.8375,B 24.8307,C -3.0008,E1 24.9569,E2 -884.6284} C_DIS
LIN {X -4.2078,Y -20.093,Z 59,A -108.0311,B 24.8313,C -2.9963,E1 24.97,E2 -889.4307} C_DIS
LIN {X -2.8194,Y -20.3349,Z 59,A -104.038,B 24.8313,C -2.9957,E1 24.981,E2 -893.4258} C_DIS
LIN {X -1.5331,Y -20.472,Z 59,A -100.264,B 24.8313,C -2.9967,E1 24.9915,E2 -897.204} C_DIS
LIN {X -0.0075,Y -20.5288,Z 59,A -95.8972,B 24.831,C -2.9982,E1 25.0037,E2 -901.5746} C_DIS
Enddeposition()
LIN {X -0.0075,Y -20.5288,Z 59,A -95.8972,B 24.831,C -2.9982,E1 25.0037,E2 -901.5746} C_DIS
Startdeposition()
$VEL.CP = VEL_PRINT
LIN {X -0.2167,Y -19.5476,Z 59,A -98.9693,B 24.831,C -2.9982,E1 24.9951,E2 -898.5027} C_DIS
LIN {X -1.926,Y -19.4536,Z 59,A -103.645,B 24.8308,C -3.0004,E1 24.9821,E2 -893.8303} C_DIS
LIN {X -3.8729,Y -19.1611,Z 59,A -110.1738,B 24.8311,C -2.9976,E1 24.9641,E2 -887.2885} C_DIS
LIN {X -5.4798,Y -18.765,Z 59,A -114.2471,B 24.8303,C -3.0049,E1 24.9532,E2 -883.2264} C_DIS
LIN {X -6.8703,Y -18.3014,Z 59,A -118.9384,B 24.8301,C -3.0063,E1 24.9408,E2 -878.5292} C_DIS
LIN {X -8.5157,Y -17.5961,Z 59,A -124.4995,B 24.8297,C -3.0104,E1 24.9267,E2 -872.9642} C_DIS
LIN {X -10.0431,Y -16.7717,Z 59,A -128.9225,B 24.8285,C -3.0205,E1 24.916,E2 -868.5523} C_DIS
LIN {X -10.9419,Y -16.1991,Z 59,A -132.5411,B 24.8282,C -3.0229,E1 24.9075,E2 -864.9277} C_DIS
LIN {X -12.3869,Y -15.1236,Z 59,A -137.6406,B 24.8271,C -3.0329,E1 24.8963,E2 -859.8333} C_DIS
LIN {X -13.5934,Y -14.0487,Z 59,A -141.9826,B 24.8258,C -3.0438,E1 24.8874,E2 -855.4998} C_DIS
LIN {X -14.5498,Y -13.0557,Z 59,A -146.4953,B 24.8251,C -3.0505,E1 24.8788,E2 -850.9832} C_DIS
LIN {X -15.5774,Y -11.8104,Z 59,A -151.1297,B 24.8238,C -3.0617,E1 24.8707,E2 -846.354} C_DIS
LIN {X -16.4479,Y -10.5648,Z 59,A -155.8492,B 24.8226,C -3.0717,E1 24.8634,E2 -841.6349} C_DIS
LIN {X -17.3433,Y -9.0188,Z 59,A -160.9951,B 24.821,C -3.0858,E1 24.8565,E2 -836.4955} C_DIS
LIN {X -18.018,Y -7.5828,Z 59,A -165.3822,B 24.8194,C -3.0995,E1 24.8515,E2 -832.1171} C_DIS
LIN {X -18.4514,Y -6.4565,Z 59,A -168.9146,B 24.8182,C -3.1095,E1 24.8481,E2 -828.5889} C_DIS
LIN {X -18.8126,Y -5.3136,Z 59,A -172.5969,B 24.8171,C -3.1192,E1 24.8451,E2 -824.9086} C_DIS
LIN {X -19.129,Y -4.0272,Z 59,A -176.3225,B 24.8156,C -3.1313,E1 24.8428,E2 -821.1901} C_DIS
LIN {X -19.3762,Y -2.5905,Z 59,A 178.5422,B 24.8144,C -3.1416,E1 24.8407,E2 -816.0487} C_DIS
LIN {X -19.5392,Y -0.607,Z 59,A 173.102,B 24.8121,C -3.1608,E1 24.8398,E2 -810.6221} C_DIS
LIN {X -19.5318,Y 0.8098,Z 59,A 169.2548,B 24.8105,C -3.1747,E1 24.84,E2 -806.7849} C_DIS
LIN {X -19.4311,Y 2.1264,Z 59,A 165.4801,B 24.809,C -3.1871,E1 24.841,E2 -803.0173} C_DIS
LIN {X -19.2044,Y 3.6522,Z 59,A 160.1598,B 24.8076,C -3.1986,E1 24.8434,E2 -797.6929} C_DIS
LIN {X -18.7985,Y 5.3633,Z 59,A 155.6044,B 24.8055,C -3.2162,E1 24.8466,E2 -793.1533} C_DIS
LIN {X -18.3888,Y 6.6332,Z 59,A 151.4491,B 24.8041,C -3.2272,E1 24.8503,E2 -789.0006} C_DIS
LIN {X -17.7859,Y 8.1125,Z 59,A 146.9613,B 24.8024,C -3.2416,E1 24.8552,E2 -784.5224} C_DIS
LIN {X -17.193,Y 9.3003,Z 59,A 143.2227,B 24.8009,C -3.2532,E1 24.86,E2 -780.7918} C_DIS
LIN {X -16.4657,Y 10.537,Z 59,A 138.8404,B 24.7996,C -3.2642,E1 24.8663,E2 -776.4132} C_DIS
LIN {X -15.8528,Y 11.4385,Z 59,A 134.4792,B 24.799,C -3.2685,E1 24.8734,E2 -772.0411} C_DIS
LIN {X -14.3973,Y 13.2236,Z 59,A 128.2814,B 24.7967,C -3.2873,E1 24.8847,E2 -765.8601} C_DIS
LIN {X -12.9926,Y 14.6062,Z 59,A 123.4514,B 24.7946,C -3.3043,E1 24.8944,E2 -761.0508} C_DIS
LIN {X -11.3798,Y 15.8949,Z 59,A 116.3336,B 24.7936,C -3.3123,E1 24.9101,E2 -753.9261} C_DIS
LIN {X -10.0103,Y 16.791,Z 59,A 111.8088,B 24.7924,C -3.3221,E1 24.9208,E2 -749.4106} C_DIS
LIN {X -8.9857,Y 17.3609,Z 59,A 108.724,B 24.7915,C -3.3294,E1 24.9284,E2 -746.3345} C_DIS
LIN {X -7.9896,Y 17.8411,Z 59,A 105.0747,B 24.7911,C -3.3322,E1 24.9377,E2 -742.6829} C_DIS
LIN {X -6.5786,Y 18.4083,Z 59,A 100.4783,B 24.7905,C -3.3372,E1 24.9497,E2 -738.089} C_DIS
LIN {X -5.1888,Y 18.8473,Z 59,A 96.5711,B 24.7896,C -3.3437,E1 24.9601,E2 -734.1906} C_DIS
LIN {X -3.9637,Y 19.1426,Z 59,A 92.7903,B 24.7893,C -3.3464,E1 24.9704,E2 -730.4115} C_DIS
LIN {X -2.8389,Y 19.3414,Z 59,A 89.3053,B 24.7891,C -3.3479,E1 24.98,E2 -726.927} C_DIS
LIN {X -1.5434,Y 19.4876,Z 59,A 85.4537,B 24.7889,C -3.3496,E1 24.9907,E2 -723.0773} C_DIS
LIN {X -0.0209,Y 19.5486,Z 59,A 81.4234,B 24.7884,C -3.3534,E1 25.0019,E2 -719.0556} C_DIS
LIN {X 1.1573,Y 19.5143,Z 59,A 77.6093,B 24.7887,C -3.3513,E1 25.0126,E2 -715.2378} C_DIS
LIN {X 2.7599,Y 19.3525,Z 59,A 72.4548,B 24.7891,C -3.3477,E1 25.0269,E2 -710.0786} C_DIS
LIN {X 4.6533,Y 18.9867,Z 59,A 66.8166,B 24.7895,C -3.3451,E1 25.0422,E2 -704.4416} C_DIS
LIN {X 6.7059,Y 18.362,Z 59,A 61.2891,B 24.7895,C -3.3455,E1 25.0569,E2 -698.9256} C_DIS
LIN {X 7.8016,Y 17.9242,Z 59,A 56.6771,B 24.7909,C -3.3336,E1 25.0688,E2 -694.2961} C_DIS
LIN {X 10.0436,Y 16.7714,Z 59,A 50.3548,B 24.7911,C -3.3319,E1 25.0842,E2 -687.9881} C_DIS
Enddeposition()
END
